LIN {X 0,Y 249.004,Z 314.463,A -85,B 0,C 180,E1 -18940.479,E2 -18940.479} C_VEL
LIN {X 0,Y 248.994,Z 314.49,A -85,B 0,C 180,E1 -18943.762,E2 -18943.762} C_VEL
LIN {X 0,Y 249.907,Z 317.142,A -85,B 0,C 180,E1 -18944.046,E2 -18944.046} C_VEL
LIN {X 0,Y 252.008,Z 319.997,A -85,B 0,C 180,E1 -18944.567,E2 -18944.567} C_VEL
LIN {X 0,Y 261.034,Z 334.136,A -85,B 0,C 180,E1 -18946.731,E2 -18946.731} C_VEL
LIN {X 0,Y 268.672,Z 348.631,A -85,B 0,C 180,E1 -18948.486,E2 -18948.486} C_VEL
LIN {X 0,Y 273.447,Z 359.161,A -85,B 0,C 180,E1 -18949.559,E2 -18949.559} C_VEL
LIN {X 0,Y 270.893,Z 419.37,A -85,B 0,C 180,E1 -18951.127,E2 -18951.127} C_VEL
LIN {X 0,Y 269.96,Z 432.258,A -85,B 0,C 180,E1 -18951.75,E2 -18951.75} C_VEL
LIN {X 0,Y 268.424,Z 444.743,A -85,B 0,C 180,E1 -18952.621,E2 -18952.621} C_VEL
LIN {X 0,Y 266.516,Z 455.493,A -85,B 0,C 180,E1 -18953.608,E2 -18953.608} C_VEL
LIN {X 0,Y 264.431,Z 466.288,A -85,B 0,C 180,E1 -18954.919,E2 -18954.919} C_VEL
LIN {X 0,Y 261.963,Z 477.569,A -85,B 0,C 180,E1 -18956.701,E2 -18956.701} C_VEL
LIN {X 0,Y 259.375,Z 487.065,A -85,B 0,C 180,E1 -18958.562,E2 -18958.562} C_VEL
LIN {X 0,Y 257.027,Z 495.055,A -85,B 0,C 180,E1 -18960.517,E2 -18960.517} C_VEL
LIN {X 0,Y 254.585,Z 502.795,A -85,B 0,C 180,E1 -18962.904,E2 -18962.904} C_VEL
LIN {X 0,Y 252.411,Z 508.966,A -85,B 0,C 180,E1 -18965.315,E2 -18965.315} C_VEL
LIN {X 0,Y 250.814,Z 513.574,A -85,B 0,C 180,E1 -18967.623,E2 -18967.623} C_VEL
LIN {X 0,Y 249.331,Z 517.523,A -85,B 0,C 180,E1 -18970.231,E2 -18970.231} C_VEL
LIN {X 0,Y 248.648,Z 519.417,A -85,B 0,C 180,E1 -18971.887,E2 -18971.887} C_VEL
LIN {X 0,Y 247.809,Z 521.57,A -85,B 0,C 180,E1 -18974.638,E2 -18974.638} C_VEL
LIN {X 0,Y 247.328,Z 522.447,A -85,B 0,C 180,E1 -18976.861,E2 -18976.861} C_VEL
LIN {X 0,Y 247.024,Z 522.665,A -85,B 0,C 180,E1 -18978.514,E2 -18978.514} C_VEL
LIN {X 0,Y 246.927,Z 522.444,A -85,B 0,C 180,E1 -18980.168,E2 -18980.168} C_VEL
LIN {X 0,Y 246.96,Z 521.821,A -85,B 0,C 180,E1 -18981.821,E2 -18981.821} C_VEL
LIN {X 0,Y 247.195,Z 520.115,A -85,B 0,C 180,E1 -18984.326,E2 -18984.326} C_VEL
LIN {X 0,Y 247.479,Z 516.49,A -85,B 0,C 180,E1 -18987.56,E2 -18987.56} C_VEL
LIN {X 0,Y 248.087,Z 512.532,A -85,B 0,C 180,E1 -18990.001,E2 -18990.001} C_VEL
LIN {X 0,Y 248.838,Z 507.454,A -85,B 0,C 180,E1 -18992.429,E2 -18992.429} C_VEL
LIN {X 0,Y 249.967,Z 501.052,A -85,B 0,C 180,E1 -18994.84,E2 -18994.84} C_VEL
LIN {X 0,Y 251.429,Z 493.077,A -85,B 0,C 180,E1 -18997.227,E2 -18997.227} C_VEL
LIN {X 0,Y 252.886,Z 484.949,A -85,B 0,C 180,E1 -18999.196,E2 -18999.196} C_VEL
LIN {X 0,Y 254.516,Z 475.048,A -85,B 0,C 180,E1 -19001.146,E2 -19001.146} C_VEL
LIN {X 0,Y 256.243,Z 463.84,A -85,B 0,C 180,E1 -19002.877,E2 -19002.877} C_VEL
LIN {X 0,Y 257.699,Z 452.872,A -85,B 0,C 180,E1 -19004.209,E2 -19004.209} C_VEL
LIN {X 0,Y 258.85,Z 440.774,A -85,B 0,C 180,E1 -19005.351,E2 -19005.351} C_VEL
LIN {X 0,Y 259.86,Z 428.037,A -85,B 0,C 180,E1 -19006.196,E2 -19006.196} C_VEL
LIN {X 0,Y 260.444,Z 414.653,A -85,B 0,C 180,E1 -19006.763,E2 -19006.763} C_VEL
LIN {X 0,Y 262.544,Z 346.789,A -85,B 0,C 180,E1 -19008.57,E2 -19008.57} C_VEL
LIN {X 0,Y 256.779,Z 331.182,A -85,B 0,C 180,E1 -19009.625,E2 -19009.625} C_VEL
LIN {X 0,Y 249.824,Z 316.729,A -85,B 0,C 180,E1 -19010.835,E2 -19010.835} C_VEL
LIN {X 0,Y 249.109,Z 314.453,A -85,B 0,C 180,E1 -19011.042,E2 -19011.042} C_VEL
LIN {X 0,Y 249.09,Z 314.446,A -85,B 0,C 180,E1 -19015.46,E2 -19015.46} C_VEL
LIN {X 0,Y 249.042,Z 314.462,A -85,B 0,C 180,E1 -19018.974,E2 -19018.974} C_VEL
LIN {X 0,Y 249.032,Z 314.463,A -85,B 0,C 180,E1 -19022.427,E2 -19022.427} C_VEL
LIN {X 0,Y 249.032,Z 314.463,A -85,B 0,C 180,E1 -19026.346,E2 -19026.346} C_VEL
LIN {X 0,Y 248.984,Z 314.465,A -85,B 0,C 180,E1 -19030.484,E2 -19030.484} C_VEL
LIN {X 0,Y 248.967,Z 314.471,A -85,B 0,C 180,E1 -19034.889,E2 -19034.889} C_VEL
LIN {X 0,Y 248.982,Z 314.46,A -85,B 0,C 180,E1 -19037.355,E2 -19037.355} C_VEL
LIN {X 0,Y 249.044,Z 314.459,A -85,B 0,C 180,E1 -19042.202,E2 -19042.202} C_VEL
LIN {X 0,Y 249.048,Z 314.45,A -85,B 0,C 180,E1 -19045.639,E2 -19045.639} C_VEL
LIN {X 0,Y 249.007,Z 314.468,A -85,B 0,C 180,E1 -19049.466,E2 -19049.466} C_VEL
LIN {X 0,Y 249.032,Z 314.458,A -85,B 0,C 180,E1 -19053.157,E2 -19053.157} C_VEL
LIN {X 0,Y 249.049,Z 314.455,A -85,B 0,C 180,E1 -19056.729,E2 -19056.729} C_VEL
LIN {X 0,Y 249.09,Z 314.456,A -85,B 0,C 180,E1 -19060.209,E2 -19060.209} C_VEL
LIN {X 0,Y 249.201,Z 314.431,A -85,B 0,C 180,E1 -19063.619,E2 -19063.619} C_VEL
LIN {X 0,Y 249.238,Z 314.436,A -85,B 0,C 180,E1 -19068.615,E2 -19068.615} C_VEL
LIN {X 0,Y 249.44,Z 314.412,A -85,B 0,C 180,E1 -19071.901,E2 -19071.901} C_VEL
LIN {X 0,Y 249.265,Z 314.416,A -85,B 0,C 180,E1 -19075.147,E2 -19075.147} C_VEL
LIN {X 0,Y 249.661,Z 314.382,A -85,B 0,C 180,E1 -19078.386,E2 -19078.386} C_VEL
LIN {X 0,Y 249.663,Z 314.384,A -85,B 0,C 180,E1 -19081.613,E2 -19081.613} C_VEL
LIN {X 0,Y 249.429,Z 314.398,A -85,B 0,C 180,E1 -19086.471,E2 -19086.471} C_VEL
LIN {X 0,Y 249.37,Z 314.418,A -85,B 0,C 180,E1 -19089.587,E2 -19089.587} C_VEL
LIN {X 0,Y 248.563,Z 314.523,A -85,B 0,C 180,E1 -19090.932,E2 -19090.932} C_VEL
LIN {X 0,Y 245.674,Z 314.891,A -85,B 0,C 180,E1 -19093.126,E2 -19093.126} C_VEL
LIN {X 0,Y 243.279,Z 315.191,A -85,B 0,C 180,E1 -19094.912,E2 -19094.912} C_VEL
LIN {X 0,Y 242.221,Z 315.317,A -85,B 0,C 180,E1 -19096.296,E2 -19096.296} C_VEL
LIN {X 0,Y 242.114,Z 315.327,A -85,B 0,C 180,E1 -19096.766,E2 -19096.766} C_VEL
LIN {X 0,Y 241.996,Z 315.339,A -85,B 0,C 180,E1 -19101.665,E2 -19101.665} C_VEL
LIN {X 0,Y 242.036,Z 315.335,A -85,B 0,C 180,E1 -19105.82,E2 -19105.82} C_VEL
LIN {X 0,Y 241.967,Z 315.344,A -85,B 0,C 180,E1 -19109.588,E2 -19109.588} C_VEL
LIN {X 0,Y 241.982,Z 315.344,A -85,B 0,C 180,E1 -19113.492,E2 -19113.492} C_VEL
LIN {X 0,Y 241.986,Z 315.343,A -85,B 0,C 180,E1 -19117.582,E2 -19117.582} C_VEL
LIN {X 0,Y 241.911,Z 315.351,A -85,B 0,C 180,E1 -19121.928,E2 -19121.928} C_VEL
LIN {X 0,Y 241.903,Z 315.35,A -85,B 0,C 180,E1 -19126.579,E2 -19126.579} C_VEL
LIN {X 0,Y 241.995,Z 315.342,A -85,B 0,C 180,E1 -19131.64,E2 -19131.64} C_VEL
LIN {X 0,Y 242.078,Z 315.472,A -85,B 0,C 180,E1 -19133.376,E2 -19133.376} C_VEL
LIN {X 0,Y 244.407,Z 325.946,A -85,B 0,C 180,E1 -19137.372,E2 -19137.372} C_VEL
LIN {X 0,Y 245.662,Z 332.102,A -85,B 0,C 180,E1 -19139.542,E2 -19139.542} C_VEL
LIN {X 0,Y 250.101,Z 344.165,A -85,B 0,C 180,E1 -19140.425,E2 -19140.425} C_VEL
LIN {X 0,Y 253.396,Z 369.809,A -85,B 0,C 180,E1 -19141.569,E2 -19141.569} C_VEL
LIN {X 0,Y 255.075,Z 385.817,A -85,B 0,C 180,E1 -19142.225,E2 -19142.225} C_VEL
LIN {X 0,Y 253.455,Z 440.891,A -85,B 0,C 180,E1 -19143.772,E2 -19143.772} C_VEL
LIN {X 0,Y 252.408,Z 454.202,A -85,B 0,C 180,E1 -19144.431,E2 -19144.431} C_VEL
LIN {X 0,Y 250.993,Z 466.976,A -85,B 0,C 180,E1 -19145.384,E2 -19145.384} C_VEL
LIN {X 0,Y 249.503,Z 478.329,A -85,B 0,C 180,E1 -19146.554,E2 -19146.554} C_VEL
LIN {X 0,Y 247.677,Z 490.055,A -85,B 0,C 180,E1 -19148.133,E2 -19148.133} C_VEL
LIN {X 0,Y 245.777,Z 500.589,A -85,B 0,C 180,E1 -19149.931,E2 -19149.931} C_VEL
LIN {X 0,Y 244.087,Z 510.234,A -85,B 0,C 180,E1 -19152.01,E2 -19152.01} C_VEL
LIN {X 0,Y 243.125,Z 516.416,A -85,B 0,C 180,E1 -19153.629,E2 -19153.629} C_VEL
LIN {X 0,Y 241.768,Z 524.334,A -85,B 0,C 180,E1 -19156.123,E2 -19156.123} C_VEL
LIN {X 0,Y 240.881,Z 529.707,A -85,B 0,C 180,E1 -19158.214,E2 -19158.214} C_VEL
LIN {X 0,Y 240.312,Z 534.946,A -85,B 0,C 180,E1 -19160.743,E2 -19160.743} C_VEL
LIN {X 0,Y 239.98,Z 538.995,A -85,B 0,C 180,E1 -19163.272,E2 -19163.272} C_VEL
LIN {X 0,Y 239.92,Z 541.078,A -85,B 0,C 180,E1 -19164.957,E2 -19164.957} C_VEL
LIN {X 0,Y 239.949,Z 542.73,A -85,B 0,C 180,E1 -19166.641,E2 -19166.641} C_VEL
LIN {X 0,Y 239.999,Z 543.969,A -85,B 0,C 180,E1 -19168.321,E2 -19168.321} C_VEL
LIN {X 0,Y 240.02,Z 544.783,A -85,B 0,C 180,E1 -19169.999,E2 -19169.999} C_VEL
LIN {X 0,Y 239.975,Z 545.159,A -85,B 0,C 180,E1 -19171.677,E2 -19171.677} C_VEL
LIN {X 0,Y 239.843,Z 544.771,A -85,B 0,C 180,E1 -19174.94,E2 -19174.94} C_VEL
LIN {X 0,Y 239.9,Z 543.946,A -85,B 0,C 180,E1 -19176.728,E2 -19176.728} C_VEL
LIN {X 0,Y 240.161,Z 542.72,A -85,B 0,C 180,E1 -19178.413,E2 -19178.413} C_VEL
LIN {X 0,Y 241.118,Z 539.053,A -85,B 0,C 180,E1 -19181.772,E2 -19181.772} C_VEL
LIN {X 0,Y 242.269,Z 535.123,A -85,B 0,C 180,E1 -19184.274,E2 -19184.274} C_VEL
LIN {X 0,Y 244.025,Z 530.087,A -85,B 0,C 180,E1 -19186.737,E2 -19186.737} C_VEL
LIN {X 0,Y 246.049,Z 523.992,A -85,B 0,C 180,E1 -19189.098,E2 -19189.098} C_VEL
LIN {X 0,Y 248.08,Z 517.373,A -85,B 0,C 180,E1 -19191.173,E2 -19191.173} C_VEL
LIN {X 0,Y 250.476,Z 509.699,A -85,B 0,C 180,E1 -19193.129,E2 -19193.129} C_VEL
LIN {X 0,Y 253.26,Z 500.391,A -85,B 0,C 180,E1 -19195.035,E2 -19195.035} C_VEL
LIN {X 0,Y 256.042,Z 490.065,A -85,B 0,C 180,E1 -19196.709,E2 -19196.709} C_VEL
LIN {X 0,Y 258.723,Z 478.628,A -85,B 0,C 180,E1 -19198.162,E2 -19198.162} C_VEL
LIN {X 0,Y 261.046,Z 466.681,A -85,B 0,C 180,E1 -19199.317,E2 -19199.317} C_VEL
LIN {X 0,Y 263.056,Z 453.416,A -85,B 0,C 180,E1 -19200.227,E2 -19200.227} C_VEL
LIN {X 0,Y 264.375,Z 440.684,A -85,B 0,C 180,E1 -19200.81,E2 -19200.81} C_VEL
LIN {X 0,Y 266.485,Z 389.159,A -85,B 0,C 180,E1 -19202.213,E2 -19202.213} C_VEL
LIN {X 0,Y 263.336,Z 367.774,A -85,B 0,C 180,E1 -19203.42,E2 -19203.42} C_VEL
LIN {X 0,Y 262.236,Z 363.038,A -85,B 0,C 180,E1 -19203.76,E2 -19203.76} C_VEL
LIN {X 0,Y 255.3,Z 347.85,A -85,B 0,C 180,E1 -19205.488,E2 -19205.488} C_VEL
LIN {X 0,Y 248.566,Z 334.814,A -85,B 0,C 180,E1 -19207.241,E2 -19207.241} C_VEL
LIN {X 0,Y 246.197,Z 330.21,A -85,B 0,C 180,E1 -19207.947,E2 -19207.947} C_VEL
LIN {X 0,Y 243.761,Z 321.533,A -85,B 0,C 180,E1 -19211.966,E2 -19211.966} C_VEL
LIN {X 0,Y 241.952,Z 315.348,A -85,B 0,C 180,E1 -19215.109,E2 -19215.109} C_VEL
LIN {X 0,Y 241.928,Z 315.343,A -85,B 0,C 180,E1 -19219.05,E2 -19219.05} C_VEL
LIN {X 0,Y 241.986,Z 315.335,A -85,B 0,C 180,E1 -19222.418,E2 -19222.418} C_VEL
LIN {X 0,Y 241.977,Z 315.34,A -85,B 0,C 180,E1 -19226.507,E2 -19226.507} C_VEL
LIN {X 0,Y 242.032,Z 315.334,A -85,B 0,C 180,E1 -19230.587,E2 -19230.587} C_VEL
LIN {X 0,Y 242.064,Z 315.331,A -85,B 0,C 180,E1 -19234.183,E2 -19234.183} C_VEL
LIN {X 0,Y 242.05,Z 315.332,A -85,B 0,C 180,E1 -19238.297,E2 -19238.297} C_VEL
LIN {X 0,Y 242.159,Z 315.311,A -85,B 0,C 180,E1 -19243.278,E2 -19243.278} C_VEL
LIN {X 0,Y 242.183,Z 315.308,A -85,B 0,C 180,E1 -19248.28,E2 -19248.28} C_VEL
LIN {X 0,Y 242.432,Z 315.277,A -85,B 0,C 180,E1 -19251.666,E2 -19251.666} C_VEL
LIN {X 0,Y 242.258,Z 315.304,A -85,B 0,C 180,E1 -19255.008,E2 -19255.008} C_VEL
LIN {X 0,Y 242.634,Z 315.26,A -85,B 0,C 180,E1 -19258.341,E2 -19258.341} C_VEL
LIN {X 0,Y 242.634,Z 315.256,A -85,B 0,C 180,E1 -19261.66,E2 -19261.66} C_VEL
LIN {X 0,Y 242.427,Z 315.284,A -85,B 0,C 180,E1 -19266.733,E2 -19266.733} C_VEL
LIN {X 0,Y 242.343,Z 315.291,A -85,B 0,C 180,E1 -19270.021,E2 -19270.021} C_VEL
LIN {X 0,Y 242.164,Z 315.319,A -85,B 0,C 180,E1 -19275.142,E2 -19275.142} C_VEL
LIN {X 0,Y 242.071,Z 315.327,A -85,B 0,C 180,E1 -19278.625,E2 -19278.625} C_VEL
LIN {X 0,Y 242.011,Z 315.333,A -85,B 0,C 180,E1 -19282.181,E2 -19282.181} C_VEL
LIN {X 0,Y 242.064,Z 315.326,A -85,B 0,C 180,E1 -19285.839,E2 -19285.839} C_VEL
LIN {X 0,Y 242.005,Z 315.334,A -85,B 0,C 180,E1 -19289.584,E2 -19289.584} C_VEL
LIN {X 0,Y 241.979,Z 315.34,A -85,B 0,C 180,E1 -19293.494,E2 -19293.494} C_VEL
LIN {X 0,Y 241.987,Z 315.336,A -85,B 0,C 180,E1 -19297.583,E2 -19297.583} C_VEL
LIN {X 0,Y 241.953,Z 315.364,A -85,B 0,C 180,E1 -19302.306,E2 -19302.306} C_VEL
LIN {X 0,Y 242.979,Z 318.216,A -85,B 0,C 180,E1 -19302.644,E2 -19302.644} C_VEL
LIN {X 0,Y 244.901,Z 320.584,A -85,B 0,C 180,E1 -19303.147,E2 -19303.147} C_VEL
LIN {X 0,Y 247.13,Z 324.018,A -85,B 0,C 180,E1 -19303.743,E2 -19303.743} C_VEL
LIN {X 0,Y 255.301,Z 336.912,A -85,B 0,C 180,E1 -19305.805,E2 -19305.805} C_VEL
LIN {X 0,Y 260.026,Z 345.326,A -85,B 0,C 180,E1 -19306.943,E2 -19306.943} C_VEL
LIN {X 0,Y 266.261,Z 358.237,A -85,B 0,C 180,E1 -19308.418,E2 -19308.418} C_VEL
LIN {X 0,Y 267.602,Z 361.247,A -85,B 0,C 180,E1 -19308.73,E2 -19308.73} C_VEL
LIN {X 0,Y 265.096,Z 418.751,A -85,B 0,C 180,E1 -19310.249,E2 -19310.249} C_VEL
LIN {X 0,Y 264.104,Z 431.812,A -85,B 0,C 180,E1 -19310.865,E2 -19310.865} C_VEL
LIN {X 0,Y 262.551,Z 444.507,A -85,B 0,C 180,E1 -19311.757,E2 -19311.757} C_VEL
LIN {X 0,Y 260.382,Z 456.275,A -85,B 0,C 180,E1 -19312.85,E2 -19312.85} C_VEL
LIN {X 0,Y 257.948,Z 468.272,A -85,B 0,C 180,E1 -19314.383,E2 -19314.383} C_VEL
LIN {X 0,Y 255.306,Z 479.371,A -85,B 0,C 180,E1 -19316.214,E2 -19316.214} C_VEL
LIN {X 0,Y 252.698,Z 488.496,A -85,B 0,C 180,E1 -19318.102,E2 -19318.102} C_VEL
LIN {X 0,Y 249.907,Z 497.336,A -85,B 0,C 180,E1 -19320.418,E2 -19320.418} C_VEL
LIN {X 0,Y 247.325,Z 504.959,A -85,B 0,C 180,E1 -19322.958,E2 -19322.958} C_VEL
LIN {X 0,Y 245.182,Z 510.763,A -85,B 0,C 180,E1 -19325.442,E2 -19325.442} C_VEL
LIN {X 0,Y 243.46,Z 515.287,A -85,B 0,C 180,E1 -19327.96,E2 -19327.96} C_VEL
LIN {X 0,Y 242.52,Z 517.656,A -85,B 0,C 180,E1 -19329.651,E2 -19329.651} C_VEL
LIN {X 0,Y 241.743,Z 519.584,A -85,B 0,C 180,E1 -19331.351,E2 -19331.351} C_VEL
LIN {X 0,Y 240.774,Z 521.944,A -85,B 0,C 180,E1 -19334.42,E2 -19334.42} C_VEL
LIN {X 0,Y 240.299,Z 522.737,A -85,B 0,C 180,E1 -19336.47,E2 -19336.47} C_VEL
LIN {X 0,Y 239.979,Z 522.985,A -85,B 0,C 180,E1 -19338.172,E2 -19338.172} C_VEL
LIN {X 0,Y 239.851,Z 522.823,A -85,B 0,C 180,E1 -19339.875,E2 -19339.875} C_VEL
LIN {X 0,Y 239.969,Z 521.251,A -85,B 0,C 180,E1 -19343.274,E2 -19343.274} C_VEL
LIN {X 0,Y 240.124,Z 519.885,A -85,B 0,C 180,E1 -19344.964,E2 -19344.964} C_VEL
LIN {X 0,Y 240.385,Z 517.019,A -85,B 0,C 180,E1 -19347.488,E2 -19347.488} C_VEL
LIN {X 0,Y 241.009,Z 513.127,A -85,B 0,C 180,E1 -19350.001,E2 -19350.001} C_VEL
LIN {X 0,Y 241.771,Z 508.125,A -85,B 0,C 180,E1 -19352.5,E2 -19352.5} C_VEL
LIN {X 0,Y 242.92,Z 501.834,A -85,B 0,C 180,E1 -19354.98,E2 -19354.98} C_VEL
LIN {X 0,Y 244.426,Z 493.956,A -85,B 0,C 180,E1 -19357.435,E2 -19357.435} C_VEL
LIN {X 0,Y 246.221,Z 484.171,A -85,B 0,C 180,E1 -19359.862,E2 -19359.862} C_VEL
LIN {X 0,Y 247.986,Z 473.94,A -85,B 0,C 180,E1 -19361.858,E2 -19361.858} C_VEL
LIN {X 0,Y 249.805,Z 462.389,A -85,B 0,C 180,E1 -19363.629,E2 -19363.629} C_VEL
LIN {X 0,Y 251.284,Z 450.994,A -85,B 0,C 180,E1 -19364.994,E2 -19364.994} C_VEL
LIN {X 0,Y 252.442,Z 439.229,A -85,B 0,C 180,E1 -19366.062,E2 -19366.062} C_VEL
LIN {X 0,Y 253.443,Z 425.644,A -85,B 0,C 180,E1 -19366.929,E2 -19366.929} C_VEL
LIN {X 0,Y 253.951,Z 413.482,A -85,B 0,C 180,E1 -19367.413,E2 -19367.413} C_VEL
LIN {X 0,Y 256.048,Z 348.219,A -85,B 0,C 180,E1 -19369.183,E2 -19369.183} C_VEL
LIN {X 0,Y 250.573,Z 333.661,A -85,B 0,C 180,E1 -19370.219,E2 -19370.219} C_VEL
LIN {X 0,Y 243.192,Z 318.383,A -85,B 0,C 180,E1 -19371.559,E2 -19371.559} C_VEL
LIN {X 0,Y 242.026,Z 315.332,A -85,B 0,C 180,E1 -19371.839,E2 -19371.839} C_VEL
LIN {X 0,Y 242.037,Z 315.326,A -85,B 0,C 180,E1 -19375.822,E2 -19375.822} C_VEL
LIN {X 0,Y 241.974,Z 315.342,A -85,B 0,C 180,E1 -19379.589,E2 -19379.589} C_VEL
LIN {X 0,Y 241.984,Z 315.342,A -85,B 0,C 180,E1 -19383.493,E2 -19383.493} C_VEL
LIN {X 0,Y 241.988,Z 315.342,A -85,B 0,C 180,E1 -19387.583,E2 -19387.583} C_VEL
LIN {X 0,Y 241.913,Z 315.345,A -85,B 0,C 180,E1 -19391.929,E2 -19391.929} C_VEL
LIN {X 0,Y 241.904,Z 315.345,A -85,B 0,C 180,E1 -19396.58,E2 -19396.58} C_VEL
LIN {X 0,Y 241.989,Z 315.341,A -85,B 0,C 180,E1 -19401.644,E2 -19401.644} C_VEL
LIN {X 0,Y 241.979,Z 315.332,A -85,B 0,C 180,E1 -19404.487,E2 -19404.487} C_VEL
LIN {X 0,Y 241.958,Z 315.343,A -85,B 0,C 180,E1 -19408.477,E2 -19408.477} C_VEL
LIN {X 0,Y 241.969,Z 315.337,A -85,B 0,C 180,E1 -19412.307,E2 -19412.307} C_VEL
LIN {X 0,Y 242.014,Z 315.327,A -85,B 0,C 180,E1 -19416.011,E2 -19416.011} C_VEL
LIN {X 0,Y 242.026,Z 315.337,A -85,B 0,C 180,E1 -19419.606,E2 -19419.606} C_VEL
LIN {X 0,Y 242.133,Z 315.314,A -85,B 0,C 180,E1 -19423.307,E2 -19423.307} C_VEL
LIN {X 0,Y 242.172,Z 315.318,A -85,B 0,C 180,E1 -19428.279,E2 -19428.279} C_VEL
LIN {X 0,Y 242.39,Z 315.29,A -85,B 0,C 180,E1 -19431.664,E2 -19431.664} C_VEL
LIN {X 0,Y 242.406,Z 315.281,A -85,B 0,C 180,E1 -19433.34,E2 -19433.34} C_VEL
LIN {X 0,Y 242.621,Z 315.257,A -85,B 0,C 180,E1 -19438.34,E2 -19438.34} C_VEL
LIN {X 0,Y 242.623,Z 315.261,A -85,B 0,C 180,E1 -19441.659,E2 -19441.659} C_VEL
LIN {X 0,Y 242.4,Z 315.273,A -85,B 0,C 180,E1 -19446.659,E2 -19446.659} C_VEL
LIN {X 0,Y 242.27,Z 315.303,A -85,B 0,C 180,E1 -19450.023,E2 -19450.023} C_VEL
LIN {X 0,Y 242.131,Z 315.323,A -85,B 0,C 180,E1 -19455.143,E2 -19455.143} C_VEL
LIN {X 0,Y 242.114,Z 315.327,A -85,B 0,C 180,E1 -19456.766,E2 -19456.766} C_VEL
LIN {X 0,Y 241.369,Z 315.417,A -85,B 0,C 180,E1 -19458.154,E2 -19458.154} C_VEL
LIN {X 0,Y 238.435,Z 315.785,A -85,B 0,C 180,E1 -19460.416,E2 -19460.416} C_VEL
LIN {X 0,Y 236.002,Z 316.087,A -85,B 0,C 180,E1 -19462.259,E2 -19462.259} C_VEL
LIN {X 0,Y 234.992,Z 316.212,A -85,B 0,C 180,E1 -19463.691,E2 -19463.691} C_VEL
LIN {X 0,Y 234.925,Z 316.22,A -85,B 0,C 180,E1 -19464.176,E2 -19464.176} C_VEL
LIN {X 0,Y 234.946,Z 316.219,A -85,B 0,C 180,E1 -19466.66,E2 -19466.66} C_VEL
LIN {X 0,Y 234.898,Z 316.226,A -85,B 0,C 180,E1 -19470.572,E2 -19470.572} C_VEL
LIN {X 0,Y 234.928,Z 316.223,A -85,B 0,C 180,E1 -19474.638,E2 -19474.638} C_VEL
LIN {X 0,Y 234.914,Z 316.225,A -85,B 0,C 180,E1 -19478.934,E2 -19478.934} C_VEL
LIN {X 0,Y 234.856,Z 316.232,A -85,B 0,C 180,E1 -19483.493,E2 -19483.493} C_VEL
LIN {X 0,Y 234.856,Z 316.227,A -85,B 0,C 180,E1 -19486.505,E2 -19486.505} C_VEL
LIN {X 0,Y 234.92,Z 316.224,A -85,B 0,C 180,E1 -19491.078,E2 -19491.078} C_VEL
LIN {X 0,Y 234.996,Z 316.343,A -85,B 0,C 180,E1 -19492.726,E2 -19492.726} C_VEL
LIN {X 0,Y 236.957,Z 324.925,A -85,B 0,C 180,E1 -19496.146,E2 -19496.146} C_VEL
LIN {X 0,Y 238.377,Z 331.628,A -85,B 0,C 180,E1 -19498.654,E2 -19498.654} C_VEL
LIN {X 0,Y 243.925,Z 346.675,A -85,B 0,C 180,E1 -19499.81,E2 -19499.81} C_VEL
LIN {X 0,Y 246.998,Z 371.172,A -85,B 0,C 180,E1 -19500.936,E2 -19500.936} C_VEL
LIN {X 0,Y 248.563,Z 386.873,A -85,B 0,C 180,E1 -19501.595,E2 -19501.595} C_VEL
LIN {X 0,Y 246.918,Z 440.487,A -85,B 0,C 180,E1 -19503.137,E2 -19503.137} C_VEL
LIN {X 0,Y 245.853,Z 453.828,A -85,B 0,C 180,E1 -19503.812,E2 -19503.812} C_VEL
LIN {X 0,Y 244.402,Z 466.616,A -85,B 0,C 180,E1 -19504.788,E2 -19504.788} C_VEL
LIN {X 0,Y 242.713,Z 478.774,A -85,B 0,C 180,E1 -19506.084,E2 -19506.084} C_VEL
LIN {X 0,Y 240.829,Z 490.358,A -85,B 0,C 180,E1 -19507.704,E2 -19507.704} C_VEL
LIN {X 0,Y 238.881,Z 500.782,A -85,B 0,C 180,E1 -19509.55,E2 -19509.55} C_VEL
LIN {X 0,Y 237.309,Z 509.477,A -85,B 0,C 180,E1 -19511.478,E2 -19511.478} C_VEL
LIN {X 0,Y 236.304,Z 515.701,A -85,B 0,C 180,E1 -19513.142,E2 -19513.142} C_VEL
LIN {X 0,Y 234.858,Z 523.708,A -85,B 0,C 180,E1 -19515.706,E2 -19515.706} C_VEL
LIN {X 0,Y 233.878,Z 529.113,A -85,B 0,C 180,E1 -19517.856,E2 -19517.856} C_VEL
LIN {X 0,Y 233.26,Z 534.412,A -85,B 0,C 180,E1 -19520.46,E2 -19520.46} C_VEL
LIN {X 0,Y 232.904,Z 538.51,A -85,B 0,C 180,E1 -19523.066,E2 -19523.066} C_VEL
LIN {X 0,Y 232.841,Z 540.747,A -85,B 0,C 180,E1 -19524.914,E2 -19524.914} C_VEL
LIN {X 0,Y 232.927,Z 543.568,A -85,B 0,C 180,E1 -19528.27,E2 -19528.27} C_VEL
LIN {X 0,Y 232.948,Z 544.417,A -85,B 0,C 180,E1 -19529.999,E2 -19529.999} C_VEL
LIN {X 0,Y 232.902,Z 544.819,A -85,B 0,C 180,E1 -19531.728,E2 -19531.728} C_VEL
LIN {X 0,Y 232.764,Z 544.439,A -85,B 0,C 180,E1 -19535.196,E2 -19535.196} C_VEL
LIN {X 0,Y 232.821,Z 543.673,A -85,B 0,C 180,E1 -19536.934,E2 -19536.934} C_VEL
LIN {X 0,Y 233.109,Z 542.481,A -85,B 0,C 180,E1 -19538.669,E2 -19538.669} C_VEL
LIN {X 0,Y 234.134,Z 538.858,A -85,B 0,C 180,E1 -19542.128,E2 -19542.128} C_VEL
LIN {X 0,Y 235.375,Z 534.973,A -85,B 0,C 180,E1 -19544.701,E2 -19544.701} C_VEL
LIN {X 0,Y 237.19,Z 529.987,A -85,B 0,C 180,E1 -19547.235,E2 -19547.235} C_VEL
LIN {X 0,Y 239.675,Z 522.86,A -85,B 0,C 180,E1 -19550.044,E2 -19550.044} C_VEL
LIN {X 0,Y 242.401,Z 514.502,A -85,B 0,C 180,E1 -19552.591,E2 -19552.591} C_VEL
LIN {X 0,Y 245.099,Z 506.308,A -85,B 0,C 180,E1 -19554.567,E2 -19554.567} C_VEL
LIN {X 0,Y 248.093,Z 496.337,A -85,B 0,C 180,E1 -19556.497,E2 -19556.497} C_VEL
LIN {X 0,Y 251.097,Z 485.084,A -85,B 0,C 180,E1 -19558.184,E2 -19558.184} C_VEL
LIN {X 0,Y 253.596,Z 474.083,A -85,B 0,C 180,E1 -19559.465,E2 -19559.465} C_VEL
LIN {X 0,Y 255.897,Z 461.901,A -85,B 0,C 180,E1 -19560.535,E2 -19560.535} C_VEL
LIN {X 0,Y 257.7,Z 448.878,A -85,B 0,C 180,E1 -19561.339,E2 -19561.339} C_VEL
LIN {X 0,Y 258.819,Z 435.274,A -85,B 0,C 180,E1 -19561.874,E2 -19561.874} C_VEL
LIN {X 0,Y 260.742,Z 390.727,A -85,B 0,C 180,E1 -19563.07,E2 -19563.07} C_VEL
LIN {X 0,Y 258.298,Z 373.078,A -85,B 0,C 180,E1 -19564.079,E2 -19564.079} C_VEL
LIN {X 0,Y 257.011,Z 366.357,A -85,B 0,C 180,E1 -19564.533,E2 -19564.533} C_VEL
LIN {X 0,Y 249.894,Z 350.731,A -85,B 0,C 180,E1 -19566.391,E2 -19566.391} C_VEL
LIN {X 0,Y 243.803,Z 338.95,A -85,B 0,C 180,E1 -19568.053,E2 -19568.053} C_VEL
LIN {X 0,Y 241.067,Z 334.042,A -85,B 0,C 180,E1 -19568.827,E2 -19568.827} C_VEL
LIN {X 0,Y 238.84,Z 329.792,A -85,B 0,C 180,E1 -19569.526,E2 -19569.526} C_VEL
LIN {X 0,Y 236.48,Z 321.57,A -85,B 0,C 180,E1 -19573.574,E2 -19573.574} C_VEL
LIN {X 0,Y 234.877,Z 316.222,A -85,B 0,C 180,E1 -19576.512,E2 -19576.512} C_VEL
LIN {X 0,Y 234.915,Z 316.22,A -85,B 0,C 180,E1 -19581.078,E2 -19581.078} C_VEL
LIN {X 0,Y 234.927,Z 316.212,A -85,B 0,C 180,E1 -19585.362,E2 -19585.362} C_VEL
LIN {X 0,Y 234.927,Z 316.215,A -85,B 0,C 180,E1 -19589.432,E2 -19589.432} C_VEL
LIN {X 0,Y 234.99,Z 316.211,A -85,B 0,C 180,E1 -19593.794,E2 -19593.794} C_VEL
LIN {X 0,Y 235.008,Z 316.202,A -85,B 0,C 180,E1 -19598.97,E2 -19598.97} C_VEL
LIN {X 0,Y 235.093,Z 316.192,A -85,B 0,C 180,E1 -19603.059,E2 -19603.059} C_VEL
LIN {X 0,Y 235.127,Z 316.197,A -85,B 0,C 180,E1 -19606.166,E2 -19606.166} C_VEL
LIN {X 0,Y 235.387,Z 316.156,A -85,B 0,C 180,E1 -19611.415,E2 -19611.415} C_VEL
LIN {X 0,Y 235.402,Z 316.157,A -85,B 0,C 180,E1 -19613.142,E2 -19613.142} C_VEL
LIN {X 0,Y 235.593,Z 316.137,A -85,B 0,C 180,E1 -19618.291,E2 -19618.291} C_VEL
LIN {X 0,Y 235.593,Z 316.133,A -85,B 0,C 180,E1 -19621.71,E2 -19621.71} C_VEL
LIN {X 0,Y 235.403,Z 316.161,A -85,B 0,C 180,E1 -19626.859,E2 -19626.859} C_VEL
LIN {X 0,Y 235.25,Z 316.176,A -85,B 0,C 180,E1 -19630.326,E2 -19630.326} C_VEL
LIN {X 0,Y 235.111,Z 316.198,A -85,B 0,C 180,E1 -19635.607,E2 -19635.607} C_VEL
LIN {X 0,Y 235.006,Z 316.211,A -85,B 0,C 180,E1 -19639.206,E2 -19639.206} C_VEL
LIN {X 0,Y 234.959,Z 316.216,A -85,B 0,C 180,E1 -19642.884,E2 -19642.884} C_VEL
LIN {X 0,Y 234.966,Z 316.215,A -85,B 0,C 180,E1 -19646.658,E2 -19646.658} C_VEL
LIN {X 0,Y 234.92,Z 316.221,A -85,B 0,C 180,E1 -19650.57,E2 -19650.57} C_VEL
LIN {X 0,Y 234.928,Z 316.216,A -85,B 0,C 180,E1 -19654.639,E2 -19654.639} C_VEL
LIN {X 0,Y 234.94,Z 316.213,A -85,B 0,C 180,E1 -19658.946,E2 -19658.946} C_VEL
LIN {X 0,Y 234.895,Z 316.22,A -85,B 0,C 180,E1 -19660.705,E2 -19660.705} C_VEL
LIN {X 0,Y 235.921,Z 319.13,A -85,B 0,C 180,E1 -19661.084,E2 -19661.084} C_VEL
LIN {X 0,Y 238.055,Z 321.599,A -85,B 0,C 180,E1 -19661.682,E2 -19661.682} C_VEL
LIN {X 0,Y 240.192,Z 324.893,A -85,B 0,C 180,E1 -19662.298,E2 -19662.298} C_VEL
LIN {X 0,Y 248.569,Z 337.793,A -85,B 0,C 180,E1 -19664.552,E2 -19664.552} C_VEL
LIN {X 0,Y 254.628,Z 348.265,A -85,B 0,C 180,E1 -19666.087,E2 -19666.087} C_VEL
LIN {X 0,Y 261.078,Z 361.737,A -85,B 0,C 180,E1 -19667.685,E2 -19667.685} C_VEL
LIN {X 0,Y 261.812,Z 363.458,A -85,B 0,C 180,E1 -19667.866,E2 -19667.866} C_VEL
LIN {X 0,Y 259.259,Z 419.591,A -85,B 0,C 180,E1 -19669.379,E2 -19669.379} C_VEL
LIN {X 0,Y 258.219,Z 432.619,A -85,B 0,C 180,E1 -19670.019,E2 -19670.019} C_VEL
LIN {X 0,Y 256.541,Z 445.449,A -85,B 0,C 180,E1 -19670.945,E2 -19670.945} C_VEL
LIN {X 0,Y 254.296,Z 457.063,A -85,B 0,C 180,E1 -19672.055,E2 -19672.055} C_VEL
LIN {X 0,Y 251.755,Z 468.945,A -85,B 0,C 180,E1 -19673.616,E2 -19673.616} C_VEL
LIN {X 0,Y 249.234,Z 479.16,A -85,B 0,C 180,E1 -19675.334,E2 -19675.334} C_VEL
LIN {X 0,Y 246.548,Z 488.186,A -85,B 0,C 180,E1 -19677.208,E2 -19677.208} C_VEL
LIN {X 0,Y 243.921,Z 496.222,A -85,B 0,C 180,E1 -19679.291,E2 -19679.291} C_VEL
LIN {X 0,Y 241.314,Z 503.742,A -85,B 0,C 180,E1 -19681.755,E2 -19681.755} C_VEL
LIN {X 0,Y 238.59,Z 510.77,A -85,B 0,C 180,E1 -19684.716,E2 -19684.716} C_VEL
LIN {X 0,Y 236.742,Z 515.378,A -85,B 0,C 180,E1 -19687.3,E2 -19687.3} C_VEL
LIN {X 0,Y 235.736,Z 517.789,A -85,B 0,C 180,E1 -19689.039,E2 -19689.039} C_VEL
LIN {X 0,Y 234.882,Z 519.75,A -85,B 0,C 180,E1 -19690.785,E2 -19690.785} C_VEL
LIN {X 0,Y 234.227,Z 521.285,A -85,B 0,C 180,E1 -19692.54,E2 -19692.54} C_VEL
LIN {X 0,Y 233.709,Z 522.362,A -85,B 0,C 180,E1 -19694.299,E2 -19694.299} C_VEL
LIN {X 0,Y 233.28,Z 523.026,A -85,B 0,C 180,E1 -19696.055,E2 -19696.055} C_VEL
LIN {X 0,Y 232.793,Z 523.189,A -85,B 0,C 180,E1 -19699.565,E2 -19699.565} C_VEL
LIN {X 0,Y 232.77,Z 522.638,A -85,B 0,C 180,E1 -19701.318,E2 -19701.318} C_VEL
LIN {X 0,Y 233.032,Z 520.678,A -85,B 0,C 180,E1 -19704.42,E2 -19704.42} C_VEL
LIN {X 0,Y 233.294,Z 517.547,A -85,B 0,C 180,E1 -19707.411,E2 -19707.411} C_VEL
LIN {X 0,Y 233.929,Z 513.721,A -85,B 0,C 180,E1 -19710.001,E2 -19710.001} C_VEL
LIN {X 0,Y 234.705,Z 508.789,A -85,B 0,C 180,E1 -19712.575,E2 -19712.575} C_VEL
LIN {X 0,Y 235.873,Z 502.589,A -85,B 0,C 180,E1 -19715.129,E2 -19715.129} C_VEL
LIN {X 0,Y 237.399,Z 494.84,A -85,B 0,C 180,E1 -19717.657,E2 -19717.657} C_VEL
LIN {X 0,Y 239.257,Z 485.162,A -85,B 0,C 180,E1 -19720.152,E2 -19720.152} C_VEL
LIN {X 0,Y 241.089,Z 475.138,A -85,B 0,C 180,E1 -19722.202,E2 -19722.202} C_VEL
LIN {X 0,Y 242.952,Z 463.777,A -85,B 0,C 180,E1 -19724.021,E2 -19724.021} C_VEL
LIN {X 0,Y 244.514,Z 452.643,A -85,B 0,C 180,E1 -19725.42,E2 -19725.42} C_VEL
LIN {X 0,Y 245.681,Z 441.411,A -85,B 0,C 180,E1 -19726.517,E2 -19726.517} C_VEL
LIN {X 0,Y 246.746,Z 428.675,A -85,B 0,C 180,E1 -19727.403,E2 -19727.403} C_VEL
LIN {X 0,Y 247.397,Z 415.273,A -85,B 0,C 180,E1 -19727.996,E2 -19727.996} C_VEL
LIN {X 0,Y 249.692,Z 350.118,A -85,B 0,C 180,E1 -19729.8,E2 -19729.8} C_VEL
LIN {X 0,Y 244.479,Z 336.371,A -85,B 0,C 180,E1 -19730.823,E2 -19730.823} C_VEL
LIN {X 0,Y 237.593,Z 322.121,A -85,B 0,C 180,E1 -19732.127,E2 -19732.127} C_VEL
LIN {X 0,Y 235.094,Z 317.005,A -85,B 0,C 180,E1 -19732.622,E2 -19732.622} C_VEL
LIN {X 0,Y 234.958,Z 316.214,A -85,B 0,C 180,E1 -19732.682,E2 -19732.682} C_VEL
LIN {X 0,Y 234.95,Z 316.212,A -85,B 0,C 180,E1 -19736.661,E2 -19736.661} C_VEL
LIN {X 0,Y 234.904,Z 316.223,A -85,B 0,C 180,E1 -19740.573,E2 -19740.573} C_VEL
LIN {X 0,Y 234.93,Z 316.221,A -85,B 0,C 180,E1 -19744.639,E2 -19744.639} C_VEL
LIN {X 0,Y 234.917,Z 316.223,A -85,B 0,C 180,E1 -19748.935,E2 -19748.935} C_VEL
LIN {X 0,Y 234.858,Z 316.23,A -85,B 0,C 180,E1 -19753.494,E2 -19753.494} C_VEL
LIN {X 0,Y 234.857,Z 316.222,A -85,B 0,C 180,E1 -19756.506,E2 -19756.506} C_VEL
LIN {X 0,Y 234.923,Z 316.22,A -85,B 0,C 180,E1 -19761.079,E2 -19761.079} C_VEL
LIN {X 0,Y 234.927,Z 316.207,A -85,B 0,C 180,E1 -19765.361,E2 -19765.361} C_VEL
LIN {X 0,Y 234.904,Z 316.224,A -85,B 0,C 180,E1 -19769.428,E2 -19769.428} C_VEL
LIN {X 0,Y 234.95,Z 316.202,A -85,B 0,C 180,E1 -19773.818,E2 -19773.818} C_VEL
LIN {X 0,Y 234.994,Z 316.211,A -85,B 0,C 180,E1 -19778.968,E2 -19778.968} C_VEL
LIN {X 0,Y 235.069,Z 316.194,A -85,B 0,C 180,E1 -19783.086,E2 -19783.086} C_VEL
LIN {X 0,Y 235.105,Z 316.194,A -85,B 0,C 180,E1 -19787.921,E2 -19787.921} C_VEL
LIN {X 0,Y 235.324,Z 316.169,A -85,B 0,C 180,E1 -19791.412,E2 -19791.412} C_VEL
LIN {X 0,Y 235.358,Z 316.158,A -85,B 0,C 180,E1 -19793.14,E2 -19793.14} C_VEL
LIN {X 0,Y 235.581,Z 316.133,A -85,B 0,C 180,E1 -19798.29,E2 -19798.29} C_VEL
LIN {X 0,Y 235.581,Z 316.138,A -85,B 0,C 180,E1 -19801.709,E2 -19801.709} C_VEL
LIN {X 0,Y 235.351,Z 316.151,A -85,B 0,C 180,E1 -19806.86,E2 -19806.86} C_VEL
LIN {X 0,Y 235.216,Z 316.184,A -85,B 0,C 180,E1 -19810.327,E2 -19810.327} C_VEL
LIN {X 0,Y 235.078,Z 316.201,A -85,B 0,C 180,E1 -19815.608,E2 -19815.608} C_VEL
LIN {X 0,Y 234.974,Z 316.215,A -85,B 0,C 180,E1 -19819.208,E2 -19819.208} C_VEL
LIN {X 0,Y 234.941,Z 316.219,A -85,B 0,C 180,E1 -19822.885,E2 -19822.885} C_VEL
LIN {X 0,Y 234.925,Z 316.22,A -85,B 0,C 180,E1 -19824.176,E2 -19824.176} C_VEL
LIN {X 0,Y 234.302,Z 316.304,A -85,B 0,C 180,E1 -19825.606,E2 -19825.606} C_VEL
LIN {X 0,Y 231.475,Z 316.663,A -85,B 0,C 180,E1 -19827.939,E2 -19827.939} C_VEL
LIN {X 0,Y 229.028,Z 316.965,A -85,B 0,C 180,E1 -19829.841,E2 -19829.841} C_VEL
LIN {X 0,Y 227.949,Z 317.093,A -85,B 0,C 180,E1 -19831.317,E2 -19831.317} C_VEL
LIN {X 0,Y 227.847,Z 317.102,A -85,B 0,C 180,E1 -19831.818,E2 -19831.818} C_VEL
LIN {X 0,Y 227.868,Z 317.101,A -85,B 0,C 180,E1 -19835.874,E2 -19835.874} C_VEL
LIN {X 0,Y 227.803,Z 317.108,A -85,B 0,C 180,E1 -19840.381,E2 -19840.381} C_VEL
LIN {X 0,Y 227.813,Z 317.109,A -85,B 0,C 180,E1 -19845.198,E2 -19845.198} C_VEL
LIN {X 0,Y 227.803,Z 317.102,A -85,B 0,C 180,E1 -19849.617,E2 -19849.617} C_VEL
LIN {X 0,Y 227.927,Z 317.241,A -85,B 0,C 180,E1 -19852.046,E2 -19852.046} C_VEL
LIN {X 0,Y 230.123,Z 326.647,A -85,B 0,C 180,E1 -19855.934,E2 -19855.934} C_VEL
LIN {X 0,Y 231.134,Z 331.305,A -85,B 0,C 180,E1 -19857.714,E2 -19857.714} C_VEL
LIN {X 0,Y 237.692,Z 348.612,A -85,B 0,C 180,E1 -19859.136,E2 -19859.136} C_VEL
LIN {X 0,Y 240.966,Z 375.412,A -85,B 0,C 180,E1 -19860.402,E2 -19860.402} C_VEL
LIN {X 0,Y 242.099,Z 387.123,A -85,B 0,C 180,E1 -19860.907,E2 -19860.907} C_VEL
LIN {X 0,Y 240.412,Z 440.082,A -85,B 0,C 180,E1 -19862.466,E2 -19862.466} C_VEL
LIN {X 0,Y 239.327,Z 453.454,A -85,B 0,C 180,E1 -19863.159,E2 -19863.159} C_VEL
LIN {X 0,Y 237.835,Z 466.255,A -85,B 0,C 180,E1 -19864.159,E2 -19864.159} C_VEL
LIN {X 0,Y 236.216,Z 477.624,A -85,B 0,C 180,E1 -19865.383,E2 -19865.383} C_VEL
LIN {X 0,Y 234.356,Z 488.034,A -85,B 0,C 180,E1 -19866.82,E2 -19866.82} C_VEL
LIN {X 0,Y 232.362,Z 498.811,A -85,B 0,C 180,E1 -19868.717,E2 -19868.717} C_VEL
LIN {X 0,Y 230.599,Z 508.522,A -85,B 0,C 180,E1 -19870.872,E2 -19870.872} C_VEL
LIN {X 0,Y 229.151,Z 516.482,A -85,B 0,C 180,E1 -19873.059,E2 -19873.059} C_VEL
LIN {X 0,Y 227.712,Z 524.224,A -85,B 0,C 180,E1 -19875.704,E2 -19875.704} C_VEL
LIN {X 0,Y 226.626,Z 530.435,A -85,B 0,C 180,E1 -19878.37,E2 -19878.37} C_VEL
LIN {X 0,Y 226.071,Z 535.366,A -85,B 0,C 180,E1 -19881.057,E2 -19881.057} C_VEL
LIN {X 0,Y 225.765,Z 539.143,A -85,B 0,C 180,E1 -19883.744,E2 -19883.744} C_VEL
LIN {X 0,Y 225.75,Z 541.881,A -85,B 0,C 180,E1 -19886.429,E2 -19886.429} C_VEL
LIN {X 0,Y 225.855,Z 543.166,A -85,B 0,C 180,E1 -19888.216,E2 -19888.216} C_VEL
LIN {X 0,Y 225.878,Z 544.043,A -85,B 0,C 180,E1 -19889.999,E2 -19889.999} C_VEL
LIN {X 0,Y 225.807,Z 544.478,A -85,B 0,C 180,E1 -19891.782,E2 -19891.782} C_VEL
LIN {X 0,Y 225.683,Z 544.139,A -85,B 0,C 180,E1 -19895.359,E2 -19895.359} C_VEL
LIN {X 0,Y 225.768,Z 543.394,A -85,B 0,C 180,E1 -19897.152,E2 -19897.152} C_VEL
LIN {X 0,Y 226.053,Z 542.241,A -85,B 0,C 180,E1 -19898.942,E2 -19898.942} C_VEL
LIN {X 0,Y 226.532,Z 540.656,A -85,B 0,C 180,E1 -19900.727,E2 -19900.727} C_VEL
LIN {X 0,Y 227.498,Z 537.502,A -85,B 0,C 180,E1 -19903.396,E2 -19903.396} C_VEL
LIN {X 0,Y 229.091,Z 533.315,A -85,B 0,C 180,E1 -19906.026,E2 -19906.026} C_VEL
LIN {X 0,Y 231.493,Z 526.964,A -85,B 0,C 180,E1 -19909.047,E2 -19909.047} C_VEL
LIN {X 0,Y 233.931,Z 520.078,A -85,B 0,C 180,E1 -19911.593,E2 -19911.593} C_VEL
LIN {X 0,Y 236.916,Z 511.508,A -85,B 0,C 180,E1 -19914.071,E2 -19914.071} C_VEL
LIN {X 0,Y 239.898,Z 502.735,A -85,B 0,C 180,E1 -19916.067,E2 -19916.067} C_VEL
LIN {X 0,Y 243.119,Z 491.964,A -85,B 0,C 180,E1 -19918.017,E2 -19918.017} C_VEL
LIN {X 0,Y 246.017,Z 481.191,A -85,B 0,C 180,E1 -19919.522,E2 -19919.522} C_VEL
LIN {X 0,Y 248.232,Z 471.112,A -85,B 0,C 180,E1 -19920.637,E2 -19920.637} C_VEL
LIN {X 0,Y 250.422,Z 459.139,A -85,B 0,C 180,E1 -19921.631,E2 -19921.631} C_VEL
LIN {X 0,Y 252.214,Z 445.898,A -85,B 0,C 180,E1 -19922.398,E2 -19922.398} C_VEL
LIN {X 0,Y 253.159,Z 432.955,A -85,B 0,C 180,E1 -19922.874,E2 -19922.874} C_VEL
LIN {X 0,Y 255.04,Z 391.459,A -85,B 0,C 180,E1 -19923.998,E2 -19923.998} C_VEL
LIN {X 0,Y 251.992,Z 370.16,A -85,B 0,C 180,E1 -19925.292,E2 -19925.292} C_VEL
LIN {X 0,Y 245.657,Z 355.801,A -85,B 0,C 180,E1 -19927.031,E2 -19927.031} C_VEL
LIN {X 0,Y 239.357,Z 343.443,A -85,B 0,C 180,E1 -19928.825,E2 -19928.825} C_VEL
LIN {X 0,Y 233.971,Z 333.825,A -85,B 0,C 180,E1 -19930.444,E2 -19930.444} C_VEL
LIN {X 0,Y 231.464,Z 329.299,A -85,B 0,C 180,E1 -19931.283,E2 -19931.283} C_VEL
LIN {X 0,Y 229.307,Z 321.887,A -85,B 0,C 180,E1 -19935.177,E2 -19935.177} C_VEL
LIN {X 0,Y 227.823,Z 317.105,A -85,B 0,C 180,E1 -19937.988,E2 -19937.988} C_VEL
LIN {X 0,Y 227.841,Z 317.096,A -85,B 0,C 180,E1 -19941.909,E2 -19941.909} C_VEL
LIN {X 0,Y 227.876,Z 317.095,A -85,B 0,C 180,E1 -19946.377,E2 -19946.377} C_VEL
LIN {X 0,Y 227.914,Z 317.093,A -85,B 0,C 180,E1 -19950.437,E2 -19950.437} C_VEL
LIN {X 0,Y 227.925,Z 317.089,A -85,B 0,C 180,E1 -19954.426,E2 -19954.426} C_VEL
LIN {X 0,Y 227.978,Z 317.084,A -85,B 0,C 180,E1 -19958.289,E2 -19958.289} C_VEL
LIN {X 0,Y 228.031,Z 317.073,A -85,B 0,C 180,E1 -19962.826,E2 -19962.826} C_VEL
LIN {X 0,Y 228.078,Z 317.075,A -85,B 0,C 180,E1 -19965.729,E2 -19965.729} C_VEL
LIN {X 0,Y 228.322,Z 317.037,A -85,B 0,C 180,E1 -19971.147,E2 -19971.147} C_VEL
LIN {X 0,Y 228.355,Z 317.033,A -85,B 0,C 180,E1 -19972.929,E2 -19972.929} C_VEL
LIN {X 0,Y 228.552,Z 317.014,A -85,B 0,C 180,E1 -19978.238,E2 -19978.238} C_VEL
LIN {X 0,Y 228.552,Z 317.01,A -85,B 0,C 180,E1 -19981.763,E2 -19981.763} C_VEL
LIN {X 0,Y 228.355,Z 317.04,A -85,B 0,C 180,E1 -19987.072,E2 -19987.072} C_VEL
LIN {X 0,Y 228.169,Z 317.059,A -85,B 0,C 180,E1 -19990.651,E2 -19990.651} C_VEL
LIN {X 0,Y 228.055,Z 317.076,A -85,B 0,C 180,E1 -19996.103,E2 -19996.103} C_VEL
LIN {X 0,Y 227.94,Z 317.091,A -85,B 0,C 180,E1 -19999.826,E2 -19999.826} C_VEL
LIN {X 0,Y 227.912,Z 317.095,A -85,B 0,C 180,E1 -20003.633,E2 -20003.633} C_VEL
LIN {X 0,Y 227.877,Z 317.098,A -85,B 0,C 180,E1 -20007.557,E2 -20007.557} C_VEL
LIN {X 0,Y 227.865,Z 317.094,A -85,B 0,C 180,E1 -20011.624,E2 -20011.624} C_VEL
LIN {X 0,Y 227.879,Z 317.091,A -85,B 0,C 180,E1 -20015.873,E2 -20015.873} C_VEL
LIN {X 0,Y 227.88,Z 317.112,A -85,B 0,C 180,E1 -20018.994,E2 -20018.994} C_VEL
LIN {X 0,Y 228.882,Z 319.947,A -85,B 0,C 180,E1 -20019.381,E2 -20019.381} C_VEL
LIN {X 0,Y 231.077,Z 322.489,A -85,B 0,C 180,E1 -20020.05,E2 -20020.05} C_VEL
LIN {X 0,Y 233.112,Z 325.729,A -85,B 0,C 180,E1 -20020.691,E2 -20020.691} C_VEL
LIN {X 0,Y 234.509,Z 327.633,A -85,B 0,C 180,E1 -20021.106,E2 -20021.106} C_VEL
LIN {X 0,Y 240.422,Z 336.561,A -85,B 0,C 180,E1 -20022.815,E2 -20022.815} C_VEL
LIN {X 0,Y 247.646,Z 348.284,A -85,B 0,C 180,E1 -20024.763,E2 -20024.763} C_VEL
LIN {X 0,Y 254.068,Z 361.041,A -85,B 0,C 180,E1 -20026.441,E2 -20026.441} C_VEL
LIN {X 0,Y 256.133,Z 365.666,A -85,B 0,C 180,E1 -20026.972,E2 -20026.972} C_VEL
LIN {X 0,Y 253.502,Z 420.071,A -85,B 0,C 180,E1 -20028.457,E2 -20028.457} C_VEL
LIN {X 0,Y 252.411,Z 433.059,A -85,B 0,C 180,E1 -20029.108,E2 -20029.108} C_VEL
LIN {X 0,Y 250.561,Z 446.386,A -85,B 0,C 180,E1 -20030.088,E2 -20030.088} C_VEL
LIN {X 0,Y 248.26,Z 457.832,A -85,B 0,C 180,E1 -20031.221,E2 -20031.221} C_VEL
LIN {X 0,Y 245.61,Z 469.625,A -85,B 0,C 180,E1 -20032.81,E2 -20032.81} C_VEL
LIN {X 0,Y 242.871,Z 480.184,A -85,B 0,C 180,E1 -20034.639,E2 -20034.639} C_VEL
LIN {X 0,Y 239.906,Z 489.589,A -85,B 0,C 180,E1 -20036.684,E2 -20036.684} C_VEL
LIN {X 0,Y 236.728,Z 498.794,A -85,B 0,C 180,E1 -20039.246,E2 -20039.246} C_VEL
LIN {X 0,Y 234.033,Z 505.908,A -85,B 0,C 180,E1 -20041.774,E2 -20041.774} C_VEL
LIN {X 0,Y 232.036,Z 510.766,A -85,B 0,C 180,E1 -20043.95,E2 -20043.95} C_VEL
LIN {X 0,Y 230.074,Z 515.45,A -85,B 0,C 180,E1 -20046.604,E2 -20046.604} C_VEL
LIN {X 0,Y 228.969,Z 517.924,A -85,B 0,C 180,E1 -20048.389,E2 -20048.389} C_VEL
LIN {X 0,Y 228.041,Z 519.916,A -85,B 0,C 180,E1 -20050.185,E2 -20050.185} C_VEL
LIN {X 0,Y 227.319,Z 521.483,A -85,B 0,C 180,E1 -20051.992,E2 -20051.992} C_VEL
LIN {X 0,Y 226.701,Z 522.688,A -85,B 0,C 180,E1 -20053.956,E2 -20053.956} C_VEL
LIN {X 0,Y 225.928,Z 523.622,A -85,B 0,C 180,E1 -20057.424,E2 -20057.424} C_VEL
LIN {X 0,Y 225.73,Z 523.541,A -85,B 0,C 180,E1 -20059.235,E2 -20059.235} C_VEL
LIN {X 0,Y 225.673,Z 523.047,A -85,B 0,C 180,E1 -20061.043,E2 -20061.043} C_VEL
LIN {X 0,Y 225.96,Z 520.98,A -85,B 0,C 180,E1 -20064.446,E2 -20064.446} C_VEL
LIN {X 0,Y 226.207,Z 518.075,A -85,B 0,C 180,E1 -20067.33,E2 -20067.33} C_VEL
LIN {X 0,Y 226.829,Z 514.316,A -85,B 0,C 180,E1 -20070.001,E2 -20070.001} C_VEL
LIN {X 0,Y 227.639,Z 509.454,A -85,B 0,C 180,E1 -20072.655,E2 -20072.655} C_VEL
LIN {X 0,Y 228.82,Z 503.333,A -85,B 0,C 180,E1 -20075.288,E2 -20075.288} C_VEL
LIN {X 0,Y 230.381,Z 495.719,A -85,B 0,C 180,E1 -20077.891,E2 -20077.891} C_VEL
LIN {X 0,Y 232.299,Z 486.153,A -85,B 0,C 180,E1 -20080.46,E2 -20080.46} C_VEL
LIN {X 0,Y 234.202,Z 476.286,A -85,B 0,C 180,E1 -20082.567,E2 -20082.567} C_VEL
LIN {X 0,Y 236.113,Z 465.162,A -85,B 0,C 180,E1 -20084.436,E2 -20084.436} C_VEL
LIN {X 0,Y 237.733,Z 454.274,A -85,B 0,C 180,E1 -20085.871,E2 -20085.871} C_VEL
LIN {X 0,Y 239.053,Z 442.286,A -85,B 0,C 180,E1 -20087.098,E2 -20087.098} C_VEL
LIN {X 0,Y 240.177,Z 429.879,A -85,B 0,C 180,E1 -20088.005,E2 -20088.005} C_VEL
LIN {X 0,Y 240.833,Z 417.054,A -85,B 0,C 180,E1 -20088.614,E2 -20088.614} C_VEL
LIN {X 0,Y 243.109,Z 351.229,A -85,B 0,C 180,E1 -20090.502,E2 -20090.502} C_VEL
LIN {X 0,Y 238.221,Z 338.521,A -85,B 0,C 180,E1 -20091.501,E2 -20091.501} C_VEL
LIN {X 0,Y 231.858,Z 325.463,A -85,B 0,C 180,E1 -20092.758,E2 -20092.758} C_VEL
LIN {X 0,Y 228.146,Z 318.271,A -85,B 0,C 180,E1 -20093.516,E2 -20093.516} C_VEL
LIN {X 0,Y 227.899,Z 317.087,A -85,B 0,C 180,E1 -20093.635,E2 -20093.635} C_VEL
LIN {X 0,Y 227.86,Z 317.097,A -85,B 0,C 180,E1 -20097.56,E2 -20097.56} C_VEL
LIN {X 0,Y 227.861,Z 317.101,A -85,B 0,C 180,E1 -20101.625,E2 -20101.625} C_VEL
LIN {X 0,Y 227.87,Z 317.099,A -85,B 0,C 180,E1 -20105.875,E2 -20105.875} C_VEL
LIN {X 0,Y 227.805,Z 317.101,A -85,B 0,C 180,E1 -20110.383,E2 -20110.383} C_VEL
LIN {X 0,Y 227.815,Z 317.105,A -85,B 0,C 180,E1 -20115.199,E2 -20115.199} C_VEL
LIN {X 0,Y 227.802,Z 317.104,A -85,B 0,C 180,E1 -20119.617,E2 -20119.617} C_VEL
LIN {X 0,Y 227.869,Z 317.089,A -85,B 0,C 180,E1 -20124.125,E2 -20124.125} C_VEL
LIN {X 0,Y 227.861,Z 317.099,A -85,B 0,C 180,E1 -20128.376,E2 -20128.376} C_VEL
LIN {X 0,Y 227.853,Z 317.095,A -85,B 0,C 180,E1 -20132.44,E2 -20132.44} C_VEL
LIN {X 0,Y 227.887,Z 317.089,A -85,B 0,C 180,E1 -20136.364,E2 -20136.364} C_VEL
LIN {X 0,Y 227.929,Z 317.092,A -85,B 0,C 180,E1 -20140.173,E2 -20140.173} C_VEL
LIN {X 0,Y 228.035,Z 317.061,A -85,B 0,C 180,E1 -20143.896,E2 -20143.896} C_VEL
LIN {X 0,Y 228.063,Z 317.068,A -85,B 0,C 180,E1 -20147.542,E2 -20147.542} C_VEL
LIN {X 0,Y 228.262,Z 317.048,A -85,B 0,C 180,E1 -20151.144,E2 -20151.144} C_VEL
LIN {X 0,Y 228.311,Z 317.036,A -85,B 0,C 180,E1 -20152.927,E2 -20152.927} C_VEL
LIN {X 0,Y 228.539,Z 317.009,A -85,B 0,C 180,E1 -20158.237,E2 -20158.237} C_VEL
LIN {X 0,Y 228.539,Z 317.016,A -85,B 0,C 180,E1 -20161.762,E2 -20161.762} C_VEL
LIN {X 0,Y 228.304,Z 317.029,A -85,B 0,C 180,E1 -20167.073,E2 -20167.073} C_VEL
LIN {X 0,Y 228.146,Z 317.067,A -85,B 0,C 180,E1 -20170.651,E2 -20170.651} C_VEL
LIN {X 0,Y 228.037,Z 317.076,A -85,B 0,C 180,E1 -20174.273,E2 -20174.273} C_VEL
LIN {X 0,Y 227.934,Z 317.09,A -85,B 0,C 180,E1 -20177.959,E2 -20177.959} C_VEL
LIN {X 0,Y 227.908,Z 317.096,A -85,B 0,C 180,E1 -20182.312,E2 -20182.312} C_VEL
LIN {X 0,Y 227.925,Z 317.094,A -85,B 0,C 180,E1 -20186.591,E2 -20186.591} C_VEL
LIN {X 0,Y 227.873,Z 317.1,A -85,B 0,C 180,E1 -20190.278,E2 -20190.278} C_VEL
LIN {X 0,Y 227.847,Z 317.102,A -85,B 0,C 180,E1 -20191.818,E2 -20191.818} C_VEL
LIN {X 0,Y 227.148,Z 317.193,A -85,B 0,C 180,E1 -20193.293,E2 -20193.293} C_VEL
LIN {X 0,Y 224.309,Z 317.545,A -85,B 0,C 180,E1 -20195.702,E2 -20195.702} C_VEL
LIN {X 0,Y 221.91,Z 317.847,A -85,B 0,C 180,E1 -20197.666,E2 -20197.666} C_VEL
LIN {X 0,Y 220.87,Z 317.975,A -85,B 0,C 180,E1 -20199.19,E2 -20199.19} C_VEL
LIN {X 0,Y 220.779,Z 317.984,A -85,B 0,C 180,E1 -20199.707,E2 -20199.707} C_VEL
LIN {X 0,Y 220.756,Z 317.986,A -85,B 0,C 180,E1 -20204.458,E2 -20204.458} C_VEL
LIN {X 0,Y 220.75,Z 317.986,A -85,B 0,C 180,E1 -20208.041,E2 -20208.041} C_VEL
LIN {X 0,Y 220.852,Z 318.132,A -85,B 0,C 180,E1 -20211.314,E2 -20211.314} C_VEL
LIN {X 0,Y 223.187,Z 327.782,A -85,B 0,C 180,E1 -20215.471,E2 -20215.471} C_VEL
LIN {X 0,Y 223.779,Z 330.724,A -85,B 0,C 180,E1 -20216.674,E2 -20216.674} C_VEL
LIN {X 0,Y 231.438,Z 350.397,A -85,B 0,C 180,E1 -20218.413,E2 -20218.413} C_VEL
LIN {X 0,Y 234.3,Z 373.706,A -85,B 0,C 180,E1 -20219.563,E2 -20219.563} C_VEL
LIN {X 0,Y 235.652,Z 388.329,A -85,B 0,C 180,E1 -20220.214,E2 -20220.214} C_VEL
LIN {X 0,Y 233.877,Z 440.777,A -85,B 0,C 180,E1 -20221.812,E2 -20221.812} C_VEL
LIN {X 0,Y 232.667,Z 454.574,A -85,B 0,C 180,E1 -20222.57,E2 -20222.57} C_VEL
LIN {X 0,Y 231.142,Z 466.957,A -85,B 0,C 180,E1 -20223.596,E2 -20223.596} C_VEL
LIN {X 0,Y 229.193,Z 479.648,A -85,B 0,C 180,E1 -20225.061,E2 -20225.061} C_VEL
LIN {X 0,Y 227.185,Z 490.953,A -85,B 0,C 180,E1 -20226.769,E2 -20226.769} C_VEL
LIN {X 0,Y 225.123,Z 501.1,A -85,B 0,C 180,E1 -20228.72,E2 -20228.72} C_VEL
LIN {X 0,Y 223.149,Z 510.741,A -85,B 0,C 180,E1 -20231.061,E2 -20231.061} C_VEL
LIN {X 0,Y 222.351,Z 515.769,A -85,B 0,C 180,E1 -20232.525,E2 -20232.525} C_VEL
LIN {X 0,Y 220.79,Z 523.602,A -85,B 0,C 180,E1 -20235.246,E2 -20235.246} C_VEL
LIN {X 0,Y 219.633,Z 529.869,A -85,B 0,C 180,E1 -20237.994,E2 -20237.994} C_VEL
LIN {X 0,Y 219.023,Z 534.849,A -85,B 0,C 180,E1 -20240.766,E2 -20240.766} C_VEL
LIN {X 0,Y 218.7,Z 538.675,A -85,B 0,C 180,E1 -20243.541,E2 -20243.541} C_VEL
LIN {X 0,Y 218.658,Z 541.456,A -85,B 0,C 180,E1 -20246.313,E2 -20246.313} C_VEL
LIN {X 0,Y 218.761,Z 542.763,A -85,B 0,C 180,E1 -20248.158,E2 -20248.158} C_VEL
LIN {X 0,Y 218.808,Z 543.662,A -85,B 0,C 180,E1 -20249.999,E2 -20249.999} C_VEL
LIN {X 0,Y 218.713,Z 544.136,A -85,B 0,C 180,E1 -20251.84,E2 -20251.84} C_VEL
LIN {X 0,Y 218.586,Z 543.837,A -85,B 0,C 180,E1 -20255.534,E2 -20255.534} C_VEL
LIN {X 0,Y 219.018,Z 541.999,A -85,B 0,C 180,E1 -20259.231,E2 -20259.231} C_VEL
LIN {X 0,Y 219.526,Z 540.44,A -85,B 0,C 180,E1 -20261.073,E2 -20261.073} C_VEL
LIN {X 0,Y 220.567,Z 537.333,A -85,B 0,C 180,E1 -20263.825,E2 -20263.825} C_VEL
LIN {X 0,Y 222.265,Z 533.196,A -85,B 0,C 180,E1 -20266.533,E2 -20266.533} C_VEL
LIN {X 0,Y 224.791,Z 526.898,A -85,B 0,C 180,E1 -20269.638,E2 -20269.638} C_VEL
LIN {X 0,Y 227.329,Z 520.072,A -85,B 0,C 180,E1 -20272.253,E2 -20272.253} C_VEL
LIN {X 0,Y 230.453,Z 511.606,A -85,B 0,C 180,E1 -20274.791,E2 -20274.791} C_VEL
LIN {X 0,Y 233.554,Z 502.918,A -85,B 0,C 180,E1 -20276.831,E2 -20276.831} C_VEL
LIN {X 0,Y 236.881,Z 492.251,A -85,B 0,C 180,E1 -20278.823,E2 -20278.823} C_VEL
LIN {X 0,Y 239.877,Z 481.656,A -85,B 0,C 180,E1 -20280.356,E2 -20280.356} C_VEL
LIN {X 0,Y 242.601,Z 469.845,A -85,B 0,C 180,E1 -20281.672,E2 -20281.672} C_VEL
LIN {X 0,Y 244.876,Z 457.585,A -85,B 0,C 180,E1 -20282.677,E2 -20282.677} C_VEL
LIN {X 0,Y 246.594,Z 444.702,A -85,B 0,C 180,E1 -20283.418,E2 -20283.418} C_VEL
LIN {X 0,Y 247.584,Z 430.91,A -85,B 0,C 180,E1 -20283.901,E2 -20283.901} C_VEL
LIN {X 0,Y 249.343,Z 391.66,A -85,B 0,C 180,E1 -20285,E2 -20285} C_VEL
LIN {X 0,Y 246.573,Z 372.646,A -85,B 0,C 180,E1 -20286.218,E2 -20286.218} C_VEL
LIN {X 0,Y 239.521,Z 356.86,A -85,B 0,C 180,E1 -20288.257,E2 -20288.257} C_VEL
LIN {X 0,Y 232.88,Z 343.991,A -85,B 0,C 180,E1 -20290.274,E2 -20290.274} C_VEL
LIN {X 0,Y 228.828,Z 337.092,A -85,B 0,C 180,E1 -20291.56,E2 -20291.56} C_VEL
LIN {X 0,Y 226.716,Z 333.476,A -85,B 0,C 180,E1 -20292.26,E2 -20292.26} C_VEL
LIN {X 0,Y 224.317,Z 329.413,A -85,B 0,C 180,E1 -20293.082,E2 -20293.082} C_VEL
LIN {X 0,Y 224.09,Z 328.861,A -85,B 0,C 180,E1 -20293.184,E2 -20293.184} C_VEL
LIN {X 0,Y 221.786,Z 321.509,A -85,B 0,C 180,E1 -20297.392,E2 -20297.392} C_VEL
LIN {X 0,Y 220.794,Z 317.976,A -85,B 0,C 180,E1 -20299.612,E2 -20299.612} C_VEL
LIN {X 0,Y 220.821,Z 317.972,A -85,B 0,C 180,E1 -20302.792,E2 -20302.792} C_VEL
LIN {X 0,Y 220.814,Z 317.976,A -85,B 0,C 180,E1 -20307.244,E2 -20307.244} C_VEL
LIN {X 0,Y 220.832,Z 317.967,A -85,B 0,C 180,E1 -20311.486,E2 -20311.486} C_VEL
LIN {X 0,Y 220.867,Z 317.961,A -85,B 0,C 180,E1 -20315.565,E2 -20315.565} C_VEL
LIN {X 0,Y 220.896,Z 317.958,A -85,B 0,C 180,E1 -20319.515,E2 -20319.515} C_VEL
LIN {X 0,Y 221.013,Z 317.945,A -85,B 0,C 180,E1 -20323.37,E2 -20323.37} C_VEL
LIN {X 0,Y 221.109,Z 317.938,A -85,B 0,C 180,E1 -20329.006,E2 -20329.006} C_VEL
LIN {X 0,Y 221.292,Z 317.911,A -85,B 0,C 180,E1 -20332.702,E2 -20332.702} C_VEL
LIN {X 0,Y 221.51,Z 317.891,A -85,B 0,C 180,E1 -20338.182,E2 -20338.182} C_VEL
LIN {X 0,Y 221.51,Z 317.888,A -85,B 0,C 180,E1 -20341.819,E2 -20341.819} C_VEL
LIN {X 0,Y 221.308,Z 317.917,A -85,B 0,C 180,E1 -20347.298,E2 -20347.298} C_VEL
LIN {X 0,Y 221.114,Z 317.94,A -85,B 0,C 180,E1 -20350.995,E2 -20350.995} C_VEL
LIN {X 0,Y 221.014,Z 317.948,A -85,B 0,C 180,E1 -20356.631,E2 -20356.631} C_VEL
LIN {X 0,Y 220.89,Z 317.965,A -85,B 0,C 180,E1 -20360.487,E2 -20360.487} C_VEL
LIN {X 0,Y 220.865,Z 317.968,A -85,B 0,C 180,E1 -20364.436,E2 -20364.436} C_VEL
LIN {X 0,Y 220.825,Z 317.97,A -85,B 0,C 180,E1 -20368.516,E2 -20368.516} C_VEL
LIN {X 0,Y 220.815,Z 317.97,A -85,B 0,C 180,E1 -20372.757,E2 -20372.757} C_VEL
LIN {X 0,Y 220.834,Z 317.975,A -85,B 0,C 180,E1 -20377.074,E2 -20377.074} C_VEL
LIN {X 0,Y 221.705,Z 320.607,A -85,B 0,C 180,E1 -20377.463,E2 -20377.463} C_VEL
LIN {X 0,Y 223.577,Z 322.771,A -85,B 0,C 180,E1 -20378.091,E2 -20378.091} C_VEL
LIN {X 0,Y 224.378,Z 323.798,A -85,B 0,C 180,E1 -20378.359,E2 -20378.359} C_VEL
LIN {X 0,Y 226.571,Z 327.029,A -85,B 0,C 180,E1 -20379.094,E2 -20379.094} C_VEL
LIN {X 0,Y 228.114,Z 329.334,A -85,B 0,C 180,E1 -20379.599,E2 -20379.599} C_VEL
LIN {X 0,Y 232.928,Z 336.149,A -85,B 0,C 180,E1 -20381.089,E2 -20381.089} C_VEL
LIN {X 0,Y 241.655,Z 350.197,A -85,B 0,C 180,E1 -20383.616,E2 -20383.616} C_VEL
LIN {X 0,Y 246.445,Z 359.181,A -85,B 0,C 180,E1 -20384.935,E2 -20384.935} C_VEL
LIN {X 0,Y 250.475,Z 367.844,A -85,B 0,C 180,E1 -20386.027,E2 -20386.027} C_VEL
LIN {X 0,Y 247.826,Z 420.428,A -85,B 0,C 180,E1 -20387.487,E2 -20387.487} C_VEL
LIN {X 0,Y 246.637,Z 433.82,A -85,B 0,C 180,E1 -20388.176,E2 -20388.176} C_VEL
LIN {X 0,Y 244.655,Z 447.315,A -85,B 0,C 180,E1 -20389.194,E2 -20389.194} C_VEL
LIN {X 0,Y 242.283,Z 458.591,A -85,B 0,C 180,E1 -20390.346,E2 -20390.346} C_VEL
LIN {X 0,Y 239.517,Z 470.304,A -85,B 0,C 180,E1 -20391.963,E2 -20391.963} C_VEL
LIN {X 0,Y 236.661,Z 480.799,A -85,B 0,C 180,E1 -20393.829,E2 -20393.829} C_VEL
LIN {X 0,Y 233.869,Z 489.311,A -85,B 0,C 180,E1 -20395.706,E2 -20395.706} C_VEL
LIN {X 0,Y 230.535,Z 498.483,A -85,B 0,C 180,E1 -20398.274,E2 -20398.274} C_VEL
LIN {X 0,Y 227.663,Z 505.831,A -85,B 0,C 180,E1 -20400.91,E2 -20400.91} C_VEL
LIN {X 0,Y 225.513,Z 510.763,A -85,B 0,C 180,E1 -20403.137,E2 -20403.137} C_VEL
LIN {X 0,Y 223.417,Z 515.52,A -85,B 0,C 180,E1 -20405.863,E2 -20405.863} C_VEL
LIN {X 0,Y 221.722,Z 519.125,A -85,B 0,C 180,E1 -20408.623,E2 -20408.623} C_VEL
LIN {X 0,Y 220.434,Z 521.684,A -85,B 0,C 180,E1 -20411.409,E2 -20411.409} C_VEL
LIN {X 0,Y 219.679,Z 523.057,A -85,B 0,C 180,E1 -20413.695,E2 -20413.695} C_VEL
LIN {X 0,Y 218.891,Z 523.942,A -85,B 0,C 180,E1 -20417.013,E2 -20417.013} C_VEL
LIN {X 0,Y 218.598,Z 523.446,A -85,B 0,C 180,E1 -20420.751,E2 -20420.751} C_VEL
LIN {X 0,Y 218.646,Z 522.565,A -85,B 0,C 180,E1 -20422.614,E2 -20422.614} C_VEL
LIN {X 0,Y 218.889,Z 521.28,A -85,B 0,C 180,E1 -20424.474,E2 -20424.474} C_VEL
LIN {X 0,Y 219.119,Z 518.601,A -85,B 0,C 180,E1 -20427.244,E2 -20427.244} C_VEL
LIN {X 0,Y 219.712,Z 514.91,A -85,B 0,C 180,E1 -20430.001,E2 -20430.001} C_VEL
LIN {X 0,Y 220.575,Z 510.115,A -85,B 0,C 180,E1 -20432.741,E2 -20432.741} C_VEL
LIN {X 0,Y 221.767,Z 504.072,A -85,B 0,C 180,E1 -20435.457,E2 -20435.457} C_VEL
LIN {X 0,Y 223.371,Z 496.56,A -85,B 0,C 180,E1 -20438.141,E2 -20438.141} C_VEL
LIN {X 0,Y 225.014,Z 488.882,A -85,B 0,C 180,E1 -20440.347,E2 -20440.347} C_VEL
LIN {X 0,Y 227.089,Z 478.46,A -85,B 0,C 180,E1 -20442.74,E2 -20442.74} C_VEL
LIN {X 0,Y 229.056,Z 467.846,A -85,B 0,C 180,E1 -20444.664,E2 -20444.664} C_VEL
LIN {X 0,Y 230.749,Z 457.578,A -85,B 0,C 180,E1 -20446.137,E2 -20446.137} C_VEL
LIN {X 0,Y 232.21,Z 445.378,A -85,B 0,C 180,E1 -20447.505,E2 -20447.505} C_VEL
LIN {X 0,Y 233.504,Z 432.511,A -85,B 0,C 180,E1 -20448.538,E2 -20448.538} C_VEL
LIN {X 0,Y 234.259,Z 420.108,A -85,B 0,C 180,E1 -20449.214,E2 -20449.214} C_VEL
LIN {X 0,Y 236.789,Z 353.668,A -85,B 0,C 180,E1 -20451.171,E2 -20451.171} C_VEL
LIN {X 0,Y 234.105,Z 345.758,A -85,B 0,C 180,E1 -20451.771,E2 -20451.771} C_VEL
LIN {X 0,Y 227.512,Z 331.49,A -85,B 0,C 180,E1 -20453.136,E2 -20453.136} C_VEL
LIN {X 0,Y 221.036,Z 318.952,A -85,B 0,C 180,E1 -20454.516,E2 -20454.516} C_VEL
LIN {X 0,Y 220.843,Z 317.959,A -85,B 0,C 180,E1 -20454.627,E2 -20454.627} C_VEL
LIN {X 0,Y 220.809,Z 317.976,A -85,B 0,C 180,E1 -20458.519,E2 -20458.519} C_VEL
LIN {X 0,Y 220.817,Z 317.979,A -85,B 0,C 180,E1 -20462.757,E2 -20462.757} C_VEL
LIN {X 0,Y 220.807,Z 317.98,A -85,B 0,C 180,E1 -20467.276,E2 -20467.276} C_VEL
LIN {X 0,Y 220.753,Z 317.98,A -85,B 0,C 180,E1 -20471.958,E2 -20471.958} C_VEL
LIN {X 0,Y 220.757,Z 317.98,A -85,B 0,C 180,E1 -20475.541,E2 -20475.541} C_VEL
LIN {X 0,Y 220.785,Z 317.98,A -85,B 0,C 180,E1 -20480.458,E2 -20480.458} C_VEL
LIN {X 0,Y 220.83,Z 317.974,A -85,B 0,C 180,E1 -20482.793,E2 -20482.793} C_VEL
LIN {X 0,Y 220.817,Z 317.969,A -85,B 0,C 180,E1 -20487.243,E2 -20487.243} C_VEL
LIN {X 0,Y 220.806,Z 317.978,A -85,B 0,C 180,E1 -20491.481,E2 -20491.481} C_VEL
LIN {X 0,Y 220.838,Z 317.957,A -85,B 0,C 180,E1 -20495.561,E2 -20495.561} C_VEL
LIN {X 0,Y 220.883,Z 317.971,A -85,B 0,C 180,E1 -20499.512,E2 -20499.512} C_VEL
LIN {X 0,Y 220.996,Z 317.942,A -85,B 0,C 180,E1 -20503.368,E2 -20503.368} C_VEL
LIN {X 0,Y 221.068,Z 317.945,A -85,B 0,C 180,E1 -20509.003,E2 -20509.003} C_VEL
LIN {X 0,Y 221.248,Z 317.916,A -85,B 0,C 180,E1 -20512.7,E2 -20512.7} C_VEL
LIN {X 0,Y 221.472,Z 317.888,A -85,B 0,C 180,E1 -20518.181,E2 -20518.181} C_VEL
LIN {X 0,Y 221.473,Z 317.896,A -85,B 0,C 180,E1 -20521.818,E2 -20521.818} C_VEL
LIN {X 0,Y 221.242,Z 317.909,A -85,B 0,C 180,E1 -20527.3,E2 -20527.3} C_VEL
LIN {X 0,Y 221.066,Z 317.948,A -85,B 0,C 180,E1 -20530.996,E2 -20530.996} C_VEL
LIN {X 0,Y 220.982,Z 317.96,A -85,B 0,C 180,E1 -20536.632,E2 -20536.632} C_VEL
LIN {X 0,Y 220.858,Z 317.975,A -85,B 0,C 180,E1 -20540.489,E2 -20540.489} C_VEL
LIN {X 0,Y 220.849,Z 317.975,A -85,B 0,C 180,E1 -20544.437,E2 -20544.437} C_VEL
LIN {X 0,Y 220.804,Z 317.981,A -85,B 0,C 180,E1 -20548.518,E2 -20548.518} C_VEL
LIN {X 0,Y 220.814,Z 317.982,A -85,B 0,C 180,E1 -20552.756,E2 -20552.756} C_VEL
LIN {X 0,Y 220.805,Z 317.983,A -85,B 0,C 180,E1 -20557.274,E2 -20557.274} C_VEL
LIN {X 0,Y 220.779,Z 317.984,A -85,B 0,C 180,E1 -20559.707,E2 -20559.707} C_VEL
LIN {X 0,Y 220.081,Z 318.073,A -85,B 0,C 180,E1 -20561.227,E2 -20561.227} C_VEL
LIN {X 0,Y 217.189,Z 318.432,A -85,B 0,C 180,E1 -20563.707,E2 -20563.707} C_VEL
LIN {X 0,Y 214.753,Z 318.733,A -85,B 0,C 180,E1 -20565.732,E2 -20565.732} C_VEL
LIN {X 0,Y 213.726,Z 318.863,A -85,B 0,C 180,E1 -20567.306,E2 -20567.306} C_VEL
LIN {X 0,Y 213.651,Z 318.86,A -85,B 0,C 180,E1 -20567.84,E2 -20567.84} C_VEL
LIN {X 0,Y 213.755,Z 318.971,A -85,B 0,C 180,E1 -20570.504,E2 -20570.504} C_VEL
LIN {X 0,Y 215.931,Z 327.733,A -85,B 0,C 180,E1 -20574.457,E2 -20574.457} C_VEL
LIN {X 0,Y 216.571,Z 330.615,A -85,B 0,C 180,E1 -20575.606,E2 -20575.606} C_VEL
LIN {X 0,Y 222.672,Z 345.575,A -85,B 0,C 180,E1 -20577.06,E2 -20577.06} C_VEL
LIN {X 0,Y 225.541,Z 353.731,A -85,B 0,C 180,E1 -20577.749,E2 -20577.749} C_VEL
LIN {X 0,Y 228.571,Z 380.576,A -85,B 0,C 180,E1 -20579.088,E2 -20579.088} C_VEL
LIN {X 0,Y 229.261,Z 388.358,A -85,B 0,C 180,E1 -20579.444,E2 -20579.444} C_VEL
LIN {X 0,Y 227.447,Z 440.311,A -85,B 0,C 180,E1 -20581.067,E2 -20581.067} C_VEL
LIN {X 0,Y 226.206,Z 454.156,A -85,B 0,C 180,E1 -20581.844,E2 -20581.844} C_VEL
LIN {X 0,Y 224.623,Z 466.568,A -85,B 0,C 180,E1 -20582.893,E2 -20582.893} C_VEL
LIN {X 0,Y 222.767,Z 478.479,A -85,B 0,C 180,E1 -20584.29,E2 -20584.29} C_VEL
LIN {X 0,Y 220.787,Z 488.612,A -85,B 0,C 180,E1 -20585.804,E2 -20585.804} C_VEL
LIN {X 0,Y 218.654,Z 499.177,A -85,B 0,C 180,E1 -20587.809,E2 -20587.809} C_VEL
LIN {X 0,Y 216.579,Z 509.394,A -85,B 0,C 180,E1 -20590.288,E2 -20590.288} C_VEL
LIN {X 0,Y 215.201,Z 516.49,A -85,B 0,C 180,E1 -20592.416,E2 -20592.416} C_VEL
LIN {X 0,Y 213.645,Z 524.103,A -85,B 0,C 180,E1 -20595.229,E2 -20595.229} C_VEL
LIN {X 0,Y 212.368,Z 531.13,A -85,B 0,C 180,E1 -20598.546,E2 -20598.546} C_VEL
LIN {X 0,Y 211.83,Z 535.767,A -85,B 0,C 180,E1 -20601.413,E2 -20601.413} C_VEL
LIN {X 0,Y 211.573,Z 539.278,A -85,B 0,C 180,E1 -20604.28,E2 -20604.28} C_VEL
LIN {X 0,Y 211.571,Z 541.031,A -85,B 0,C 180,E1 -20606.189,E2 -20606.189} C_VEL
LIN {X 0,Y 211.67,Z 542.359,A -85,B 0,C 180,E1 -20608.096,E2 -20608.096} C_VEL
LIN {X 0,Y 211.74,Z 543.281,A -85,B 0,C 180,E1 -20609.999,E2 -20609.999} C_VEL
LIN {X 0,Y 211.622,Z 543.788,A -85,B 0,C 180,E1 -20611.902,E2 -20611.902} C_VEL
LIN {X 0,Y 211.512,Z 543.778,A -85,B 0,C 180,E1 -20614.572,E2 -20614.572} C_VEL
LIN {X 0,Y 211.631,Z 542.834,A -85,B 0,C 180,E1 -20617.632,E2 -20617.632} C_VEL
LIN {X 0,Y 211.999,Z 541.749,A -85,B 0,C 180,E1 -20619.54,E2 -20619.54} C_VEL
LIN {X 0,Y 212.513,Z 540.225,A -85,B 0,C 180,E1 -20621.444,E2 -20621.444} C_VEL
LIN {X 0,Y 213.66,Z 537.165,A -85,B 0,C 180,E1 -20624.281,E2 -20624.281} C_VEL
LIN {X 0,Y 215.459,Z 533.077,A -85,B 0,C 180,E1 -20627.07,E2 -20627.07} C_VEL
LIN {X 0,Y 218.094,Z 526.832,A -85,B 0,C 180,E1 -20630.267,E2 -20630.267} C_VEL
LIN {X 0,Y 220.743,Z 520.065,A -85,B 0,C 180,E1 -20632.954,E2 -20632.954} C_VEL
LIN {X 0,Y 224.038,Z 511.696,A -85,B 0,C 180,E1 -20635.551,E2 -20635.551} C_VEL
LIN {X 0,Y 227.249,Z 503.101,A -85,B 0,C 180,E1 -20637.638,E2 -20637.638} C_VEL
LIN {X 0,Y 230.704,Z 492.538,A -85,B 0,C 180,E1 -20639.67,E2 -20639.67} C_VEL
LIN {X 0,Y 233.808,Z 482.079,A -85,B 0,C 180,E1 -20641.231,E2 -20641.231} C_VEL
LIN {X 0,Y 236.602,Z 470.568,A -85,B 0,C 180,E1 -20642.572,E2 -20642.572} C_VEL
LIN {X 0,Y 238.957,Z 458.637,A -85,B 0,C 180,E1 -20643.592,E2 -20643.592} C_VEL
LIN {X 0,Y 240.888,Z 445.137,A -85,B 0,C 180,E1 -20644.4,E2 -20644.4} C_VEL
LIN {X 0,Y 241.891,Z 432.223,A -85,B 0,C 180,E1 -20644.89,E2 -20644.89} C_VEL
LIN {X 0,Y 243.791,Z 392.774,A -85,B 0,C 180,E1 -20646.004,E2 -20646.004} C_VEL
LIN {X 0,Y 241.403,Z 375.692,A -85,B 0,C 180,E1 -20647.129,E2 -20647.129} C_VEL
LIN {X 0,Y 234.528,Z 360.194,A -85,B 0,C 180,E1 -20649.22,E2 -20649.22} C_VEL
LIN {X 0,Y 228.455,Z 348.327,A -85,B 0,C 180,E1 -20651.162,E2 -20651.162} C_VEL
LIN {X 0,Y 223.068,Z 338.86,A -85,B 0,C 180,E1 -20652.986,E2 -20652.986} C_VEL
LIN {X 0,Y 219.46,Z 333.086,A -85,B 0,C 180,E1 -20654.268,E2 -20654.268} C_VEL
LIN {X 0,Y 216.629,Z 328.28,A -85,B 0,C 180,E1 -20655.385,E2 -20655.385} C_VEL
LIN {X 0,Y 214.735,Z 322.241,A -85,B 0,C 180,E1 -20659.113,E2 -20659.113} C_VEL
LIN {X 0,Y 213.718,Z 318.857,A -85,B 0,C 180,E1 -20661.449,E2 -20661.449} C_VEL
LIN {X 0,Y 213.753,Z 318.851,A -85,B 0,C 180,E1 -20666.018,E2 -20666.018} C_VEL
LIN {X 0,Y 213.777,Z 318.854,A -85,B 0,C 180,E1 -20670.454,E2 -20670.454} C_VEL
LIN {X 0,Y 213.8,Z 318.846,A -85,B 0,C 180,E1 -20674.702,E2 -20674.702} C_VEL
LIN {X 0,Y 213.829,Z 318.841,A -85,B 0,C 180,E1 -20678.805,E2 -20678.805} C_VEL
LIN {X 0,Y 213.94,Z 318.828,A -85,B 0,C 180,E1 -20682.804,E2 -20682.804} C_VEL
LIN {X 0,Y 213.976,Z 318.826,A -85,B 0,C 180,E1 -20686.708,E2 -20686.708} C_VEL
LIN {X 0,Y 214.193,Z 318.802,A -85,B 0,C 180,E1 -20690.558,E2 -20690.558} C_VEL
LIN {X 0,Y 214.109,Z 318.815,A -85,B 0,C 180,E1 -20694.349,E2 -20694.349} C_VEL
LIN {X 0,Y 214.443,Z 318.772,A -85,B 0,C 180,E1 -20698.122,E2 -20698.122} C_VEL
LIN {X 0,Y 214.548,Z 318.751,A -85,B 0,C 180,E1 -20700,E2 -20700} C_VEL
LIN {X 0,Y 214.443,Z 318.768,A -85,B 0,C 180,E1 -20701.879,E2 -20701.879} C_VEL
LIN {X 0,Y 214.245,Z 318.795,A -85,B 0,C 180,E1 -20707.54,E2 -20707.54} C_VEL
LIN {X 0,Y 214.045,Z 318.822,A -85,B 0,C 180,E1 -20711.362,E2 -20711.362} C_VEL
LIN {X 0,Y 213.932,Z 318.836,A -85,B 0,C 180,E1 -20715.238,E2 -20715.238} C_VEL
LIN {X 0,Y 213.866,Z 318.844,A -85,B 0,C 180,E1 -20719.185,E2 -20719.185} C_VEL
LIN {X 0,Y 213.845,Z 318.848,A -85,B 0,C 180,E1 -20723.228,E2 -20723.228} C_VEL
LIN {X 0,Y 213.827,Z 318.849,A -85,B 0,C 180,E1 -20727.451,E2 -20727.451} C_VEL
LIN {X 0,Y 213.766,Z 318.849,A -85,B 0,C 180,E1 -20731.739,E2 -20731.739} C_VEL
LIN {X 0,Y 213.768,Z 318.849,A -85,B 0,C 180,E1 -20734.941,E2 -20734.941} C_VEL
LIN {X 0,Y 214.681,Z 321.565,A -85,B 0,C 180,E1 -20735.393,E2 -20735.393} C_VEL
LIN {X 0,Y 216.699,Z 323.739,A -85,B 0,C 180,E1 -20736.133,E2 -20736.133} C_VEL
LIN {X 0,Y 217.558,Z 324.896,A -85,B 0,C 180,E1 -20736.452,E2 -20736.452} C_VEL
LIN {X 0,Y 219.501,Z 327.827,A -85,B 0,C 180,E1 -20737.172,E2 -20737.172} C_VEL
LIN {X 0,Y 220.843,Z 329.395,A -85,B 0,C 180,E1 -20737.635,E2 -20737.635} C_VEL
LIN {X 0,Y 229.183,Z 341.642,A -85,B 0,C 180,E1 -20740.41,E2 -20740.41} C_VEL
LIN {X 0,Y 237.021,Z 354.365,A -85,B 0,C 180,E1 -20742.782,E2 -20742.782} C_VEL
LIN {X 0,Y 241.801,Z 363.416,A -85,B 0,C 180,E1 -20744.16,E2 -20744.16} C_VEL
LIN {X 0,Y 244.916,Z 370.198,A -85,B 0,C 180,E1 -20745.048,E2 -20745.048} C_VEL
LIN {X 0,Y 242.243,Z 420.847,A -85,B 0,C 180,E1 -20746.476,E2 -20746.476} C_VEL
LIN {X 0,Y 240.979,Z 434.331,A -85,B 0,C 180,E1 -20747.183,E2 -20747.183} C_VEL
LIN {X 0,Y 239.031,Z 447.145,A -85,B 0,C 180,E1 -20748.161,E2 -20748.161} C_VEL
LIN {X 0,Y 236.376,Z 459.366,A -85,B 0,C 180,E1 -20749.43,E2 -20749.43} C_VEL
LIN {X 0,Y 233.564,Z 470.702,A -85,B 0,C 180,E1 -20751.028,E2 -20751.028} C_VEL
LIN {X 0,Y 230.521,Z 481.411,A -85,B 0,C 180,E1 -20752.979,E2 -20752.979} C_VEL
LIN {X 0,Y 227.286,Z 490.69,A -85,B 0,C 180,E1 -20755.108,E2 -20755.108} C_VEL
LIN {X 0,Y 223.859,Z 499.682,A -85,B 0,C 180,E1 -20757.745,E2 -20757.745} C_VEL
LIN {X 0,Y 220.871,Z 506.852,A -85,B 0,C 180,E1 -20760.45,E2 -20760.45} C_VEL
LIN {X 0,Y 218.235,Z 512.517,A -85,B 0,C 180,E1 -20763.203,E2 -20763.203} C_VEL
LIN {X 0,Y 216.056,Z 517.07,A -85,B 0,C 180,E1 -20766.115,E2 -20766.115} C_VEL
LIN {X 0,Y 214.432,Z 520.256,A -85,B 0,C 180,E1 -20768.869,E2 -20768.869} C_VEL
LIN {X 0,Y 213.562,Z 521.885,A -85,B 0,C 180,E1 -20770.788,E2 -20770.788} C_VEL
LIN {X 0,Y 212.663,Z 523.426,A -85,B 0,C 180,E1 -20773.414,E2 -20773.414} C_VEL
LIN {X 0,Y 211.874,Z 524.262,A -85,B 0,C 180,E1 -20776.575,E2 -20776.575} C_VEL
LIN {X 0,Y 211.507,Z 523.829,A -85,B 0,C 180,E1 -20780.438,E2 -20780.438} C_VEL
LIN {X 0,Y 211.554,Z 523.001,A -85,B 0,C 180,E1 -20782.365,E2 -20782.365} C_VEL
LIN {X 0,Y 211.802,Z 521.548,A -85,B 0,C 180,E1 -20784.545,E2 -20784.545} C_VEL
LIN {X 0,Y 212.139,Z 518.058,A -85,B 0,C 180,E1 -20788.103,E2 -20788.103} C_VEL
LIN {X 0,Y 212.87,Z 514.076,A -85,B 0,C 180,E1 -20790.947,E2 -20790.947} C_VEL
LIN {X 0,Y 214.043,Z 507.96,A -85,B 0,C 180,E1 -20794.238,E2 -20794.238} C_VEL
LIN {X 0,Y 215.533,Z 501.291,A -85,B 0,C 180,E1 -20797.025,E2 -20797.025} C_VEL
LIN {X 0,Y 217.346,Z 493.029,A -85,B 0,C 180,E1 -20799.775,E2 -20799.775} C_VEL
LIN {X 0,Y 219.213,Z 484.521,A -85,B 0,C 180,E1 -20802.029,E2 -20802.029} C_VEL
LIN {X 0,Y 221.331,Z 474.034,A -85,B 0,C 180,E1 -20804.247,E2 -20804.247} C_VEL
LIN {X 0,Y 223.237,Z 463.637,A -85,B 0,C 180,E1 -20805.991,E2 -20805.991} C_VEL
LIN {X 0,Y 224.939,Z 452.227,A -85,B 0,C 180,E1 -20807.502,E2 -20807.502} C_VEL
LIN {X 0,Y 226.32,Z 440.426,A -85,B 0,C 180,E1 -20808.678,E2 -20808.678} C_VEL
LIN {X 0,Y 227.484,Z 426.8,A -85,B 0,C 180,E1 -20809.633,E2 -20809.633} C_VEL
LIN {X 0,Y 228.084,Z 414.563,A -85,B 0,C 180,E1 -20810.165,E2 -20810.165} C_VEL
LIN {X 0,Y 230.309,Z 354.41,A -85,B 0,C 180,E1 -20811.96,E2 -20811.96} C_VEL
LIN {X 0,Y 226.406,Z 344.463,A -85,B 0,C 180,E1 -20812.828,E2 -20812.828} C_VEL
LIN {X 0,Y 219.605,Z 330.497,A -85,B 0,C 180,E1 -20814.303,E2 -20814.303} C_VEL
LIN {X 0,Y 213.977,Z 319.685,A -85,B 0,C 180,E1 -20815.584,E2 -20815.584} C_VEL
LIN {X 0,Y 213.825,Z 318.834,A -85,B 0,C 180,E1 -20815.688,E2 -20815.688} C_VEL
LIN {X 0,Y 213.755,Z 318.856,A -85,B 0,C 180,E1 -20819.551,E2 -20819.551} C_VEL
LIN {X 0,Y 213.759,Z 318.857,A -85,B 0,C 180,E1 -20823.983,E2 -20823.983} C_VEL
LIN {X 0,Y 213.709,Z 318.864,A -85,B 0,C 180,E1 -20828.671,E2 -20828.671} C_VEL
LIN {X 0,Y 213.706,Z 318.864,A -85,B 0,C 180,E1 -20833.655,E2 -20833.655} C_VEL
LIN {X 0,Y 213.706,Z 318.856,A -85,B 0,C 180,E1 -20836.346,E2 -20836.346} C_VEL
LIN {X 0,Y 213.708,Z 318.864,A -85,B 0,C 180,E1 -20841.329,E2 -20841.329} C_VEL
LIN {X 0,Y 213.759,Z 318.842,A -85,B 0,C 180,E1 -20846.017,E2 -20846.017} C_VEL
LIN {X 0,Y 213.754,Z 318.857,A -85,B 0,C 180,E1 -20850.449,E2 -20850.449} C_VEL
LIN {X 0,Y 213.772,Z 318.833,A -85,B 0,C 180,E1 -20854.697,E2 -20854.697} C_VEL
LIN {X 0,Y 213.803,Z 318.851,A -85,B 0,C 180,E1 -20858.802,E2 -20858.802} C_VEL
LIN {X 0,Y 213.927,Z 318.826,A -85,B 0,C 180,E1 -20862.802,E2 -20862.802} C_VEL
LIN {X 0,Y 213.942,Z 318.824,A -85,B 0,C 180,E1 -20866.705,E2 -20866.705} C_VEL
LIN {X 0,Y 214.141,Z 318.809,A -85,B 0,C 180,E1 -20870.555,E2 -20870.555} C_VEL
LIN {X 0,Y 214.079,Z 318.796,A -85,B 0,C 180,E1 -20874.347,E2 -20874.347} C_VEL
LIN {X 0,Y 214.409,Z 318.767,A -85,B 0,C 180,E1 -20878.121,E2 -20878.121} C_VEL
LIN {X 0,Y 214.517,Z 318.762,A -85,B 0,C 180,E1 -20880,E2 -20880} C_VEL
LIN {X 0,Y 214.409,Z 318.776,A -85,B 0,C 180,E1 -20881.878,E2 -20881.878} C_VEL
LIN {X 0,Y 214.184,Z 318.789,A -85,B 0,C 180,E1 -20887.541,E2 -20887.541} C_VEL
LIN {X 0,Y 213.997,Z 318.827,A -85,B 0,C 180,E1 -20891.364,E2 -20891.364} C_VEL
LIN {X 0,Y 213.903,Z 318.84,A -85,B 0,C 180,E1 -20895.239,E2 -20895.239} C_VEL
LIN {X 0,Y 213.8,Z 318.853,A -85,B 0,C 180,E1 -20899.191,E2 -20899.191} C_VEL
LIN {X 0,Y 213.798,Z 318.852,A -85,B 0,C 180,E1 -20903.232,E2 -20903.232} C_VEL
LIN {X 0,Y 213.788,Z 318.854,A -85,B 0,C 180,E1 -20907.426,E2 -20907.426} C_VEL
LIN {X 0,Y 213.762,Z 318.858,A -85,B 0,C 180,E1 -20911.738,E2 -20911.738} C_VEL
LIN {X 0,Y 213.744,Z 318.861,A -85,B 0,C 180,E1 -20916.288,E2 -20916.288} C_VEL
LIN {X 0,Y 213.7,Z 318.868,A -85,B 0,C 180,E1 -20921.128,E2 -20921.128} C_VEL
LIN {X 0,Y 213.704,Z 318.866,A -85,B 0,C 180,E1 -20923.679,E2 -20923.679} C_VEL
LIN {X 0,Y 213.651,Z 318.86,A -85,B 0,C 180,E1 -20927.84,E2 -20927.84} C_VEL
LIN {X 0,Y 213.089,Z 319.321,A -85,B 0,C 180,E1 -20928.889,E2 -20928.889} C_VEL
LIN {X 0,Y 211.291,Z 320.98,A -85,B 0,C 180,E1 -20930.187,E2 -20930.187} C_VEL
LIN {X 0,Y 208.687,Z 324.781,A -85,B 0,C 180,E1 -20932.053,E2 -20932.053} C_VEL
LIN {X 0,Y 208.507,Z 326.907,A -85,B 0,C 180,E1 -20933.01,E2 -20933.01} C_VEL
LIN {X 0,Y 209.25,Z 330.072,A -85,B 0,C 180,E1 -20934.411,E2 -20934.411} C_VEL
LIN {X 0,Y 216.697,Z 348.106,A -85,B 0,C 180,E1 -20936.283,E2 -20936.283} C_VEL
LIN {X 0,Y 219.427,Z 355.66,A -85,B 0,C 180,E1 -20936.964,E2 -20936.964} C_VEL
LIN {X 0,Y 222.357,Z 382.443,A -85,B 0,C 180,E1 -20938.343,E2 -20938.343} C_VEL
LIN {X 0,Y 222.918,Z 388.875,A -85,B 0,C 180,E1 -20938.648,E2 -20938.648} C_VEL
LIN {X 0,Y 221.052,Z 439.842,A -85,B 0,C 180,E1 -20940.278,E2 -20940.278} C_VEL
LIN {X 0,Y 219.784,Z 453.739,A -85,B 0,C 180,E1 -20941.075,E2 -20941.075} C_VEL
LIN {X 0,Y 218.141,Z 466.179,A -85,B 0,C 180,E1 -20942.149,E2 -20942.149} C_VEL
LIN {X 0,Y 216.07,Z 478.902,A -85,B 0,C 180,E1 -20943.692,E2 -20943.692} C_VEL
LIN {X 0,Y 213.834,Z 490.212,A -85,B 0,C 180,E1 -20945.483,E2 -20945.483} C_VEL
LIN {X 0,Y 211.653,Z 500.384,A -85,B 0,C 180,E1 -20947.55,E2 -20947.55} C_VEL
LIN {X 0,Y 209.632,Z 509.62,A -85,B 0,C 180,E1 -20949.914,E2 -20949.914} C_VEL
LIN {X 0,Y 208.055,Z 517.166,A -85,B 0,C 180,E1 -20952.3,E2 -20952.3} C_VEL
LIN {X 0,Y 206.487,Z 524.603,A -85,B 0,C 180,E1 -20955.209,E2 -20955.209} C_VEL
LIN {X 0,Y 205.373,Z 530.56,A -85,B 0,C 180,E1 -20958.15,E2 -20958.15} C_VEL
LIN {X 0,Y 204.781,Z 535.253,A -85,B 0,C 180,E1 -20961.115,E2 -20961.115} C_VEL
LIN {X 0,Y 204.497,Z 538.808,A -85,B 0,C 180,E1 -20964.081,E2 -20964.081} C_VEL
LIN {X 0,Y 204.476,Z 540.603,A -85,B 0,C 180,E1 -20966.057,E2 -20966.057} C_VEL
LIN {X 0,Y 204.58,Z 541.955,A -85,B 0,C 180,E1 -20968.03,E2 -20968.03} C_VEL
LIN {X 0,Y 204.672,Z 542.898,A -85,B 0,C 180,E1 -20969.999,E2 -20969.999} C_VEL
LIN {X 0,Y 204.533,Z 543.432,A -85,B 0,C 180,E1 -20971.968,E2 -20971.968} C_VEL
LIN {X 0,Y 204.438,Z 543.483,A -85,B 0,C 180,E1 -20974.486,E2 -20974.486} C_VEL
LIN {X 0,Y 204.592,Z 542.555,A -85,B 0,C 180,E1 -20977.896,E2 -20977.896} C_VEL
LIN {X 0,Y 204.962,Z 541.491,A -85,B 0,C 180,E1 -20979.871,E2 -20979.871} C_VEL
LIN {X 0,Y 205.518,Z 540.011,A -85,B 0,C 180,E1 -20981.839,E2 -20981.839} C_VEL
LIN {X 0,Y 206.746,Z 536.992,A -85,B 0,C 180,E1 -20984.769,E2 -20984.769} C_VEL
LIN {X 0,Y 208.655,Z 532.948,A -85,B 0,C 180,E1 -20987.645,E2 -20987.645} C_VEL
LIN {X 0,Y 211.422,Z 526.766,A -85,B 0,C 180,E1 -20990.936,E2 -20990.936} C_VEL
LIN {X 0,Y 214.197,Z 520.061,A -85,B 0,C 180,E1 -20993.698,E2 -20993.698} C_VEL
LIN {X 0,Y 217.648,Z 511.774,A -85,B 0,C 180,E1 -20996.358,E2 -20996.358} C_VEL
LIN {X 0,Y 220.974,Z 503.292,A -85,B 0,C 180,E1 -20998.493,E2 -20998.493} C_VEL
LIN {X 0,Y 224.58,Z 492.841,A -85,B 0,C 180,E1 -21000.564,E2 -21000.564} C_VEL
LIN {X 0,Y 227.779,Z 482.519,A -85,B 0,C 180,E1 -21002.156,E2 -21002.156} C_VEL
LIN {X 0,Y 230.672,Z 471.229,A -85,B 0,C 180,E1 -21003.518,E2 -21003.518} C_VEL
LIN {X 0,Y 233.114,Z 459.705,A -85,B 0,C 180,E1 -21004.551,E2 -21004.551} C_VEL
LIN {X 0,Y 235.187,Z 446.184,A -85,B 0,C 180,E1 -21005.4,E2 -21005.4} C_VEL
LIN {X 0,Y 236.338,Z 433.409,A -85,B 0,C 180,E1 -21005.914,E2 -21005.914} C_VEL
LIN {X 0,Y 238.318,Z 393.9,A -85,B 0,C 180,E1 -21007.054,E2 -21007.054} C_VEL
LIN {X 0,Y 236.237,Z 378.681,A -85,B 0,C 180,E1 -21008.094,E2 -21008.094} C_VEL
LIN {X 0,Y 230.217,Z 364.833,A -85,B 0,C 180,E1 -21010.024,E2 -21010.024} C_VEL
LIN {X 0,Y 224.191,Z 352.81,A -85,B 0,C 180,E1 -21012.051,E2 -21012.051} C_VEL
LIN {X 0,Y 218.761,Z 343.212,A -85,B 0,C 180,E1 -21013.984,E2 -21013.984} C_VEL
LIN {X 0,Y 215.475,Z 337.83,A -85,B 0,C 180,E1 -21015.22,E2 -21015.22} C_VEL
LIN {X 0,Y 212.459,Z 333.031,A -85,B 0,C 180,E1 -21016.41,E2 -21016.41} C_VEL
LIN {X 0,Y 209.557,Z 328.619,A -85,B 0,C 180,E1 -21017.608,E2 -21017.608} C_VEL
LIN {X 0,Y 209.137,Z 327.591,A -85,B 0,C 180,E1 -21017.919,E2 -21017.919} C_VEL
LIN {X 0,Y 207.667,Z 322.827,A -85,B 0,C 180,E1 -21021.11,E2 -21021.11} C_VEL
LIN {X 0,Y 206.691,Z 319.738,A -85,B 0,C 180,E1 -21023.485,E2 -21023.485} C_VEL
LIN {X 0,Y 206.714,Z 319.725,A -85,B 0,C 180,E1 -21028.206,E2 -21028.206} C_VEL
LIN {X 0,Y 206.763,Z 319.718,A -85,B 0,C 180,E1 -21032.096,E2 -21032.096} C_VEL
LIN {X 0,Y 206.787,Z 319.717,A -85,B 0,C 180,E1 -21036.58,E2 -21036.58} C_VEL
LIN {X 0,Y 206.87,Z 319.714,A -85,B 0,C 180,E1 -21042.197,E2 -21042.197} C_VEL
LIN {X 0,Y 206.912,Z 319.71,A -85,B 0,C 180,E1 -21046.246,E2 -21046.246} C_VEL
LIN {X 0,Y 207.13,Z 319.685,A -85,B 0,C 180,E1 -21050.233,E2 -21050.233} C_VEL
LIN {X 0,Y 207.072,Z 319.691,A -85,B 0,C 180,E1 -21054.156,E2 -21054.156} C_VEL
LIN {X 0,Y 207.38,Z 319.651,A -85,B 0,C 180,E1 -21058.058,E2 -21058.058} C_VEL
LIN {X 0,Y 207.512,Z 319.627,A -85,B 0,C 180,E1 -21060,E2 -21060} C_VEL
LIN {X 0,Y 207.38,Z 319.648,A -85,B 0,C 180,E1 -21061.943,E2 -21061.943} C_VEL
LIN {X 0,Y 207.186,Z 319.674,A -85,B 0,C 180,E1 -21067.799,E2 -21067.799} C_VEL
LIN {X 0,Y 206.981,Z 319.701,A -85,B 0,C 180,E1 -21071.756,E2 -21071.756} C_VEL
LIN {X 0,Y 206.865,Z 319.716,A -85,B 0,C 180,E1 -21075.771,E2 -21075.771} C_VEL
LIN {X 0,Y 206.797,Z 319.725,A -85,B 0,C 180,E1 -21079.868,E2 -21079.868} C_VEL
LIN {X 0,Y 206.761,Z 319.727,A -85,B 0,C 180,E1 -21084.073,E2 -21084.073} C_VEL
LIN {X 0,Y 206.735,Z 319.725,A -85,B 0,C 180,E1 -21088.421,E2 -21088.421} C_VEL
LIN {X 0,Y 206.705,Z 319.829,A -85,B 0,C 180,E1 -21092.581,E2 -21092.581} C_VEL
LIN {X 0,Y 207.544,Z 322.308,A -85,B 0,C 180,E1 -21093.024,E2 -21093.024} C_VEL
LIN {X 0,Y 209.358,Z 324.44,A -85,B 0,C 180,E1 -21093.78,E2 -21093.78} C_VEL
LIN {X 0,Y 210.375,Z 325.243,A -85,B 0,C 180,E1 -21094.171,E2 -21094.171} C_VEL
LIN {X 0,Y 212.344,Z 328.441,A -85,B 0,C 180,E1 -21094.995,E2 -21094.995} C_VEL
LIN {X 0,Y 214.063,Z 330.354,A -85,B 0,C 180,E1 -21095.646,E2 -21095.646} C_VEL
LIN {X 0,Y 216.582,Z 333.925,A -85,B 0,C 180,E1 -21096.603,E2 -21096.603} C_VEL
LIN {X 0,Y 223.356,Z 343.795,A -85,B 0,C 180,E1 -21099,E2 -21099} C_VEL
LIN {X 0,Y 231.221,Z 356.386,A -85,B 0,C 180,E1 -21101.538,E2 -21101.538} C_VEL
LIN {X 0,Y 236.725,Z 366.65,A -85,B 0,C 180,E1 -21103.212,E2 -21103.212} C_VEL
LIN {X 0,Y 239.443,Z 372.498,A -85,B 0,C 180,E1 -21104.024,E2 -21104.024} C_VEL
LIN {X 0,Y 236.737,Z 421.247,A -85,B 0,C 180,E1 -21105.417,E2 -21105.417} C_VEL
LIN {X 0,Y 235.394,Z 434.852,A -85,B 0,C 180,E1 -21106.142,E2 -21106.142} C_VEL
LIN {X 0,Y 233.502,Z 446.974,A -85,B 0,C 180,E1 -21107.082,E2 -21107.082} C_VEL
LIN {X 0,Y 230.918,Z 458.533,A -85,B 0,C 180,E1 -21108.26,E2 -21108.26} C_VEL
LIN {X 0,Y 227.874,Z 470.243,A -85,B 0,C 180,E1 -21109.896,E2 -21109.896} C_VEL
LIN {X 0,Y 224.774,Z 480.977,A -85,B 0,C 180,E1 -21111.866,E2 -21111.866} C_VEL
LIN {X 0,Y 221.382,Z 490.429,A -85,B 0,C 180,E1 -21114.036,E2 -21114.036} C_VEL
LIN {X 0,Y 217.729,Z 499.518,A -85,B 0,C 180,E1 -21116.721,E2 -21116.721} C_VEL
LIN {X 0,Y 214.583,Z 506.797,A -85,B 0,C 180,E1 -21119.494,E2 -21119.494} C_VEL
LIN {X 0,Y 211.77,Z 512.554,A -85,B 0,C 180,E1 -21122.316,E2 -21122.316} C_VEL
LIN {X 0,Y 209.876,Z 516.351,A -85,B 0,C 180,E1 -21124.709,E2 -21124.709} C_VEL
LIN {X 0,Y 207.673,Z 520.425,A -85,B 0,C 180,E1 -21128.146,E2 -21128.146} C_VEL
LIN {X 0,Y 206.711,Z 522.086,A -85,B 0,C 180,E1 -21130.125,E2 -21130.125} C_VEL
LIN {X 0,Y 205.64,Z 523.8,A -85,B 0,C 180,E1 -21133.127,E2 -21133.127} C_VEL
LIN {X 0,Y 204.877,Z 524.581,A -85,B 0,C 180,E1 -21136.107,E2 -21136.107} C_VEL
LIN {X 0,Y 204.434,Z 524.207,A -85,B 0,C 180,E1 -21140.104,E2 -21140.104} C_VEL
LIN {X 0,Y 204.441,Z 523.433,A -85,B 0,C 180,E1 -21142.098,E2 -21142.098} C_VEL
LIN {X 0,Y 204.711,Z 521.803,A -85,B 0,C 180,E1 -21144.638,E2 -21144.638} C_VEL
LIN {X 0,Y 205.049,Z 518.586,A -85,B 0,C 180,E1 -21148.037,E2 -21148.037} C_VEL
LIN {X 0,Y 205.786,Z 514.668,A -85,B 0,C 180,E1 -21150.98,E2 -21150.98} C_VEL
LIN {X 0,Y 206.826,Z 509.629,A -85,B 0,C 180,E1 -21153.898,E2 -21153.898} C_VEL
LIN {X 0,Y 208.228,Z 503.295,A -85,B 0,C 180,E1 -21156.785,E2 -21156.785} C_VEL
LIN {X 0,Y 210.026,Z 495.381,A -85,B 0,C 180,E1 -21159.633,E2 -21159.633} C_VEL
LIN {X 0,Y 212.305,Z 485.539,A -85,B 0,C 180,E1 -21162.427,E2 -21162.427} C_VEL
LIN {X 0,Y 214.508,Z 475.216,A -85,B 0,C 180,E1 -21164.711,E2 -21164.711} C_VEL
LIN {X 0,Y 216.728,Z 463.585,A -85,B 0,C 180,E1 -21166.727,E2 -21166.727} C_VEL
LIN {X 0,Y 218.494,Z 452.039,A -85,B 0,C 180,E1 -21168.278,E2 -21168.278} C_VEL
LIN {X 0,Y 219.952,Z 440.061,A -85,B 0,C 180,E1 -21169.483,E2 -21169.483} C_VEL
LIN {X 0,Y 221.073,Z 427.072,A -85,B 0,C 180,E1 -21170.409,E2 -21170.409} C_VEL
LIN {X 0,Y 221.719,Z 414.776,A -85,B 0,C 180,E1 -21170.952,E2 -21170.952} C_VEL
LIN {X 0,Y 224.017,Z 356.047,A -85,B 0,C 180,E1 -21172.742,E2 -21172.742} C_VEL
LIN {X 0,Y 220.019,Z 346.202,A -85,B 0,C 180,E1 -21173.663,E2 -21173.663} C_VEL
LIN {X 0,Y 212.498,Z 331.044,A -85,B 0,C 180,E1 -21175.383,E2 -21175.383} C_VEL
LIN {X 0,Y 207.766,Z 322.481,A -85,B 0,C 180,E1 -21176.507,E2 -21176.507} C_VEL
LIN {X 0,Y 206.778,Z 319.72,A -85,B 0,C 180,E1 -21176.82,E2 -21176.82} C_VEL
LIN {X 0,Y 206.714,Z 319.735,A -85,B 0,C 180,E1 -21181.79,E2 -21181.79} C_VEL
LIN {X 0,Y 206.704,Z 319.738,A -85,B 0,C 180,E1 -21185.312,E2 -21185.312} C_VEL
LIN {X 0,Y 206.652,Z 319.735,A -85,B 0,C 180,E1 -21190.255,E2 -21190.255} C_VEL
LIN {X 0,Y 206.634,Z 319.743,A -85,B 0,C 180,E1 -21194.417,E2 -21194.417} C_VEL
LIN {X 0,Y 206.635,Z 319.732,A -85,B 0,C 180,E1 -21198.442,E2 -21198.442} C_VEL
LIN {X 0,Y 206.672,Z 319.737,A -85,B 0,C 180,E1 -21202.258,E2 -21202.258} C_VEL
LIN {X 0,Y 206.699,Z 319.726,A -85,B 0,C 180,E1 -21207.042,E2 -21207.042} C_VEL
LIN {X 0,Y 206.713,Z 319.728,A -85,B 0,C 180,E1 -21212.128,E2 -21212.128} C_VEL
LIN {X 0,Y 206.746,Z 319.722,A -85,B 0,C 180,E1 -21216.613,E2 -21216.613} C_VEL
LIN {X 0,Y 206.873,Z 319.706,A -85,B 0,C 180,E1 -21222.196,E2 -21222.196} C_VEL
LIN {X 0,Y 206.884,Z 319.696,A -85,B 0,C 180,E1 -21226.243,E2 -21226.243} C_VEL
LIN {X 0,Y 207.085,Z 319.689,A -85,B 0,C 180,E1 -21230.23,E2 -21230.23} C_VEL
LIN {X 0,Y 207.043,Z 319.673,A -85,B 0,C 180,E1 -21234.155,E2 -21234.155} C_VEL
LIN {X 0,Y 207.348,Z 319.646,A -85,B 0,C 180,E1 -21238.057,E2 -21238.057} C_VEL
LIN {X 0,Y 207.484,Z 319.638,A -85,B 0,C 180,E1 -21240,E2 -21240} C_VEL
LIN {X 0,Y 207.349,Z 319.656,A -85,B 0,C 180,E1 -21241.942,E2 -21241.942} C_VEL
LIN {X 0,Y 207.129,Z 319.667,A -85,B 0,C 180,E1 -21247.8,E2 -21247.8} C_VEL
LIN {X 0,Y 206.919,Z 319.709,A -85,B 0,C 180,E1 -21251.758,E2 -21251.758} C_VEL
LIN {X 0,Y 206.83,Z 319.72,A -85,B 0,C 180,E1 -21255.773,E2 -21255.773} C_VEL
LIN {X 0,Y 206.721,Z 319.734,A -85,B 0,C 180,E1 -21259.875,E2 -21259.875} C_VEL
LIN {X 0,Y 206.738,Z 319.732,A -85,B 0,C 180,E1 -21264.075,E2 -21264.075} C_VEL
LIN {X 0,Y 206.691,Z 319.739,A -85,B 0,C 180,E1 -21268.426,E2 -21268.426} C_VEL
LIN {X 0,Y 206.697,Z 319.742,A -85,B 0,C 180,E1 -21272.958,E2 -21272.958} C_VEL
LIN {X 0,Y 206.671,Z 319.743,A -85,B 0,C 180,E1 -21277.741,E2 -21277.741} C_VEL
LIN {X 0,Y 206.634,Z 319.747,A -85,B 0,C 180,E1 -21281.558,E2 -21281.558} C_VEL
LIN {X 0,Y 206.632,Z 319.745,A -85,B 0,C 180,E1 -21285.582,E2 -21285.582} C_VEL
LIN {X 0,Y 206.704,Z 319.779,A -85,B 0,C 180,E1 -21289.625,E2 -21289.625} C_VEL
LIN {X 0,Y 208.507,Z 326.907,A -85,B 0,C 180,E1 -21293.01,E2 -21293.01} C_VEL
LIN {X 0,Y 209.035,Z 329.393,A -85,B 0,C 180,E1 -21293.789,E2 -21293.789} C_VEL
LIN {X 0,Y 209.772,Z 333.475,A -85,B 0,C 180,E1 -21294.466,E2 -21294.466} C_VEL
LIN {X 0,Y 210.627,Z 340.027,A -85,B 0,C 180,E1 -21295.028,E2 -21295.028} C_VEL
LIN {X 0,Y 211.855,Z 352.338,A -85,B 0,C 180,E1 -21295.7,E2 -21295.7} C_VEL
LIN {X 0,Y 212.834,Z 356.237,A -85,B 0,C 180,E1 -21296.003,E2 -21296.003} C_VEL
LIN {X 0,Y 213.514,Z 359.029,A -85,B 0,C 180,E1 -21296.214,E2 -21296.214} C_VEL
LIN {X 0,Y 216.269,Z 385.286,A -85,B 0,C 180,E1 -21297.606,E2 -21297.606} C_VEL
LIN {X 0,Y 216.542,Z 391.481,A -85,B 0,C 180,E1 -21297.873,E2 -21297.873} C_VEL
LIN {X 0,Y 214.706,Z 439.341,A -85,B 0,C 180,E1 -21299.442,E2 -21299.442} C_VEL
LIN {X 0,Y 213.406,Z 453.301,A -85,B 0,C 180,E1 -21300.26,E2 -21300.26} C_VEL
LIN {X 0,Y 211.7,Z 465.777,A -85,B 0,C 180,E1 -21301.359,E2 -21301.359} C_VEL
LIN {X 0,Y 209.653,Z 477.712,A -85,B 0,C 180,E1 -21302.822,E2 -21302.822} C_VEL
LIN {X 0,Y 207.281,Z 489.175,A -85,B 0,C 180,E1 -21304.654,E2 -21304.654} C_VEL
LIN {X 0,Y 205.009,Z 499.517,A -85,B 0,C 180,E1 -21306.78,E2 -21306.78} C_VEL
LIN {X 0,Y 202.908,Z 508.975,A -85,B 0,C 180,E1 -21309.257,E2 -21309.257} C_VEL
LIN {X 0,Y 201.283,Z 516.476,A -85,B 0,C 180,E1 -21311.684,E2 -21311.684} C_VEL
LIN {X 0,Y 199.607,Z 523.976,A -85,B 0,C 180,E1 -21314.687,E2 -21314.687} C_VEL
LIN {X 0,Y 198.376,Z 529.986,A -85,B 0,C 180,E1 -21317.726,E2 -21317.726} C_VEL
LIN {X 0,Y 197.723,Z 534.73,A -85,B 0,C 180,E1 -21320.795,E2 -21320.795} C_VEL
LIN {X 0,Y 197.41,Z 538.335,A -85,B 0,C 180,E1 -21323.868,E2 -21323.868} C_VEL
LIN {X 0,Y 197.413,Z 540.178,A -85,B 0,C 180,E1 -21325.916,E2 -21325.916} C_VEL
LIN {X 0,Y 197.492,Z 541.55,A -85,B 0,C 180,E1 -21327.959,E2 -21327.959} C_VEL
LIN {X 0,Y 197.605,Z 542.517,A -85,B 0,C 180,E1 -21329.999,E2 -21329.999} C_VEL
LIN {X 0,Y 197.446,Z 543.07,A -85,B 0,C 180,E1 -21332.039,E2 -21332.039} C_VEL
LIN {X 0,Y 197.338,Z 543.196,A -85,B 0,C 180,E1 -21334.297,E2 -21334.297} C_VEL
LIN {X 0,Y 197.527,Z 542.276,A -85,B 0,C 180,E1 -21338.181,E2 -21338.181} C_VEL
LIN {X 0,Y 198.542,Z 539.793,A -85,B 0,C 180,E1 -21342.261,E2 -21342.261} C_VEL
LIN {X 0,Y 199.858,Z 536.81,A -85,B 0,C 180,E1 -21345.291,E2 -21345.291} C_VEL
LIN {X 0,Y 201.859,Z 532.813,A -85,B 0,C 180,E1 -21348.26,E2 -21348.26} C_VEL
LIN {X 0,Y 204.784,Z 526.707,A -85,B 0,C 180,E1 -21351.648,E2 -21351.648} C_VEL
LIN {X 0,Y 207.691,Z 520.063,A -85,B 0,C 180,E1 -21354.488,E2 -21354.488} C_VEL
LIN {X 0,Y 211.318,Z 511.844,A -85,B 0,C 180,E1 -21357.211,E2 -21357.211} C_VEL
LIN {X 0,Y 214.771,Z 503.459,A -85,B 0,C 180,E1 -21359.395,E2 -21359.395} C_VEL
LIN {X 0,Y 218.517,Z 493.144,A -85,B 0,C 180,E1 -21361.508,E2 -21361.508} C_VEL
LIN {X 0,Y 221.826,Z 482.958,A -85,B 0,C 180,E1 -21363.127,E2 -21363.127} C_VEL
LIN {X 0,Y 224.812,Z 471.852,A -85,B 0,C 180,E1 -21364.513,E2 -21364.513} C_VEL
LIN {X 0,Y 227.563,Z 459.48,A -85,B 0,C 180,E1 -21365.656,E2 -21365.656} C_VEL
LIN {X 0,Y 229.703,Z 445.996,A -85,B 0,C 180,E1 -21366.515,E2 -21366.515} C_VEL
LIN {X 0,Y 230.864,Z 433.797,A -85,B 0,C 180,E1 -21367.02,E2 -21367.02} C_VEL
LIN {X 0,Y 232.926,Z 395.059,A -85,B 0,C 180,E1 -21368.153,E2 -21368.153} C_VEL
LIN {X 0,Y 231.108,Z 381.498,A -85,B 0,C 180,E1 -21369.116,E2 -21369.116} C_VEL
LIN {X 0,Y 225.356,Z 368.156,A -85,B 0,C 180,E1 -21371.068,E2 -21371.068} C_VEL
LIN {X 0,Y 219.883,Z 357.099,A -85,B 0,C 180,E1 -21373.012,E2 -21373.012} C_VEL
LIN {X 0,Y 214.853,Z 348.09,A -85,B 0,C 180,E1 -21374.898,E2 -21374.898} C_VEL
LIN {X 0,Y 210.983,Z 341.648,A -85,B 0,C 180,E1 -21376.44,E2 -21376.44} C_VEL
LIN {X 0,Y 209.054,Z 338.447,A -85,B 0,C 180,E1 -21377.249,E2 -21377.249} C_VEL
LIN {X 0,Y 205.97,Z 333.581,A -85,B 0,C 180,E1 -21378.593,E2 -21378.593} C_VEL
LIN {X 0,Y 202.179,Z 328.164,A -85,B 0,C 180,E1 -21380.329,E2 -21380.329} C_VEL
LIN {X 0,Y 201.688,Z 327.028,A -85,B 0,C 180,E1 -21380.696,E2 -21380.696} C_VEL
LIN {X 0,Y 200.068,Z 322.26,A -85,B 0,C 180,E1 -21384.321,E2 -21384.321} C_VEL
LIN {X 0,Y 199.608,Z 320.611,A -85,B 0,C 180,E1 -21385.713,E2 -21385.713} C_VEL
LIN {X 0,Y 199.69,Z 320.6,A -85,B 0,C 180,E1 -21388.135,E2 -21388.135} C_VEL
LIN {X 0,Y 199.684,Z 320.601,A -85,B 0,C 180,E1 -21392.772,E2 -21392.772} C_VEL
LIN {X 0,Y 199.743,Z 320.6,A -85,B 0,C 180,E1 -21397.23,E2 -21397.23} C_VEL
LIN {X 0,Y 199.794,Z 320.598,A -85,B 0,C 180,E1 -21401.757,E2 -21401.757} C_VEL
LIN {X 0,Y 199.847,Z 320.592,A -85,B 0,C 180,E1 -21405.75,E2 -21405.75} C_VEL
LIN {X 0,Y 200.072,Z 320.564,A -85,B 0,C 180,E1 -21409.885,E2 -21409.885} C_VEL
LIN {X 0,Y 200.035,Z 320.567,A -85,B 0,C 180,E1 -21413.95,E2 -21413.95} C_VEL
LIN {X 0,Y 200.319,Z 320.531,A -85,B 0,C 180,E1 -21417.99,E2 -21417.99} C_VEL
LIN {X 0,Y 200.477,Z 320.503,A -85,B 0,C 180,E1 -21420.001,E2 -21420.001} C_VEL
LIN {X 0,Y 200.029,Z 320.56,A -85,B 0,C 180,E1 -21424.03,E2 -21424.03} C_VEL
LIN {X 0,Y 200.129,Z 320.549,A -85,B 0,C 180,E1 -21428.076,E2 -21428.076} C_VEL
LIN {X 0,Y 199.912,Z 320.578,A -85,B 0,C 180,E1 -21432.178,E2 -21432.178} C_VEL
LIN {X 0,Y 199.804,Z 320.591,A -85,B 0,C 180,E1 -21436.344,E2 -21436.344} C_VEL
LIN {X 0,Y 199.821,Z 320.587,A -85,B 0,C 180,E1 -21438.455,E2 -21438.455} C_VEL
LIN {X 0,Y 199.735,Z 320.605,A -85,B 0,C 180,E1 -21443.818,E2 -21443.818} C_VEL
LIN {X 0,Y 199.706,Z 320.601,A -85,B 0,C 180,E1 -21448.385,E2 -21448.385} C_VEL
LIN {X 0,Y 199.674,Z 320.719,A -85,B 0,C 180,E1 -21449.886,E2 -21449.886} C_VEL
LIN {X 0,Y 200.426,Z 323.054,A -85,B 0,C 180,E1 -21450.343,E2 -21450.343} C_VEL
LIN {X 0,Y 202.35,Z 325.338,A -85,B 0,C 180,E1 -21451.253,E2 -21451.253} C_VEL
LIN {X 0,Y 203.525,Z 326.28,A -85,B 0,C 180,E1 -21451.764,E2 -21451.764} C_VEL
LIN {X 0,Y 205.576,Z 329.587,A -85,B 0,C 180,E1 -21452.721,E2 -21452.721} C_VEL
LIN {X 0,Y 207.361,Z 331.421,A -85,B 0,C 180,E1 -21453.465,E2 -21453.465} C_VEL
LIN {X 0,Y 210.016,Z 335.106,A -85,B 0,C 180,E1 -21454.577,E2 -21454.577} C_VEL
LIN {X 0,Y 216.315,Z 343.991,A -85,B 0,C 180,E1 -21457.019,E2 -21457.019} C_VEL
LIN {X 0,Y 223.655,Z 355.495,A -85,B 0,C 180,E1 -21459.611,E2 -21459.611} C_VEL
LIN {X 0,Y 229.947,Z 366.36,A -85,B 0,C 180,E1 -21461.658,E2 -21461.658} C_VEL
LIN {X 0,Y 233.986,Z 374.817,A -85,B 0,C 180,E1 -21462.94,E2 -21462.94} C_VEL
LIN {X 0,Y 231.275,Z 422.098,A -85,B 0,C 180,E1 -21464.326,E2 -21464.326} C_VEL
LIN {X 0,Y 229.878,Z 435.515,A -85,B 0,C 180,E1 -21465.061,E2 -21465.061} C_VEL
LIN {X 0,Y 227.828,Z 447.95,A -85,B 0,C 180,E1 -21466.048,E2 -21466.048} C_VEL
LIN {X 0,Y 225.145,Z 459.318,A -85,B 0,C 180,E1 -21467.241,E2 -21467.241} C_VEL
LIN {X 0,Y 222.279,Z 469.887,A -85,B 0,C 180,E1 -21468.73,E2 -21468.73} C_VEL
LIN {X 0,Y 219.108,Z 480.526,A -85,B 0,C 180,E1 -21470.693,E2 -21470.693} C_VEL
LIN {X 0,Y 215.546,Z 490.157,A -85,B 0,C 180,E1 -21472.902,E2 -21472.902} C_VEL
LIN {X 0,Y 211.702,Z 499.357,A -85,B 0,C 180,E1 -21475.644,E2 -21475.644} C_VEL
LIN {X 0,Y 208.36,Z 506.725,A -85,B 0,C 180,E1 -21478.48,E2 -21478.48} C_VEL
LIN {X 0,Y 205.387,Z 512.583,A -85,B 0,C 180,E1 -21481.378,E2 -21481.378} C_VEL
LIN {X 0,Y 203.121,Z 516.818,A -85,B 0,C 180,E1 -21484.108,E2 -21484.108} C_VEL
LIN {X 0,Y 200.953,Z 520.594,A -85,B 0,C 180,E1 -21487.376,E2 -21487.376} C_VEL
LIN {X 0,Y 199.912,Z 522.289,A -85,B 0,C 180,E1 -21489.419,E2 -21489.419} C_VEL
LIN {X 0,Y 198.418,Z 524.446,A -85,B 0,C 180,E1 -21493.54,E2 -21493.54} C_VEL
LIN {X 0,Y 197.901,Z 524.9,A -85,B 0,C 180,E1 -21495.607,E2 -21495.607} C_VEL
LIN {X 0,Y 197.342,Z 524.586,A -85,B 0,C 180,E1 -21499.744,E2 -21499.744} C_VEL
LIN {X 0,Y 197.357,Z 523.847,A -85,B 0,C 180,E1 -21501.812,E2 -21501.812} C_VEL
LIN {X 0,Y 197.626,Z 522.073,A -85,B 0,C 180,E1 -21504.718,E2 -21504.718} C_VEL
LIN {X 0,Y 198.115,Z 517.941,A -85,B 0,C 180,E1 -21508.985,E2 -21508.985} C_VEL
LIN {X 0,Y 199,Z 513.725,A -85,B 0,C 180,E1 -21512.025,E2 -21512.025} C_VEL
LIN {X 0,Y 200.373,Z 507.345,A -85,B 0,C 180,E1 -21515.536,E2 -21515.536} C_VEL
LIN {X 0,Y 202.073,Z 500.371,A -85,B 0,C 180,E1 -21518.501,E2 -21518.501} C_VEL
LIN {X 0,Y 204.186,Z 491.645,A -85,B 0,C 180,E1 -21521.416,E2 -21521.416} C_VEL
LIN {X 0,Y 206.509,Z 481.74,A -85,B 0,C 180,E1 -21524.034,E2 -21524.034} C_VEL
LIN {X 0,Y 208.667,Z 471.638,A -85,B 0,C 180,E1 -21526.134,E2 -21526.134} C_VEL
LIN {X 0,Y 210.814,Z 460.422,A -85,B 0,C 180,E1 -21527.962,E2 -21527.962} C_VEL
LIN {X 0,Y 212.572,Z 447.881,A -85,B 0,C 180,E1 -21529.559,E2 -21529.559} C_VEL
LIN {X 0,Y 214.123,Z 434.806,A -85,B 0,C 180,E1 -21530.725,E2 -21530.725} C_VEL
LIN {X 0,Y 215.092,Z 421.41,A -85,B 0,C 180,E1 -21531.534,E2 -21531.534} C_VEL
LIN {X 0,Y 217.704,Z 357.666,A -85,B 0,C 180,E1 -21533.577,E2 -21533.577} C_VEL
LIN {X 0,Y 213.1,Z 346.768,A -85,B 0,C 180,E1 -21534.683,E2 -21534.683} C_VEL
LIN {X 0,Y 204.877,Z 330.575,A -85,B 0,C 180,E1 -21536.683,E2 -21536.683} C_VEL
LIN {X 0,Y 201.174,Z 324.137,A -85,B 0,C 180,E1 -21537.616,E2 -21537.616} C_VEL
LIN {X 0,Y 199.848,Z 321.514,A -85,B 0,C 180,E1 -21537.974,E2 -21537.974} C_VEL
LIN {X 0,Y 199.676,Z 320.607,A -85,B 0,C 180,E1 -21538.089,E2 -21538.089} C_VEL
LIN {X 0,Y 199.67,Z 320.613,A -85,B 0,C 180,E1 -21542.353,E2 -21542.353} C_VEL
LIN {X 0,Y 199.622,Z 320.618,A -85,B 0,C 180,E1 -21546.765,E2 -21546.765} C_VEL
LIN {X 0,Y 199.599,Z 320.618,A -85,B 0,C 180,E1 -21549.332,E2 -21549.332} C_VEL
LIN {X 0,Y 199.571,Z 320.618,A -85,B 0,C 180,E1 -21552.308,E2 -21552.308} C_VEL
LIN {X 0,Y 199.581,Z 320.62,A -85,B 0,C 180,E1 -21555.228,E2 -21555.228} C_VEL
LIN {X 0,Y 199.573,Z 320.609,A -85,B 0,C 180,E1 -21558.002,E2 -21558.002} C_VEL
LIN {X 0,Y 199.601,Z 320.619,A -85,B 0,C 180,E1 -21560.773,E2 -21560.773} C_VEL
LIN {X 0,Y 199.615,Z 320.6,A -85,B 0,C 180,E1 -21565.713,E2 -21565.713} C_VEL
LIN {X 0,Y 199.691,Z 320.607,A -85,B 0,C 180,E1 -21568.134,E2 -21568.134} C_VEL
LIN {X 0,Y 199.643,Z 320.606,A -85,B 0,C 180,E1 -21572.765,E2 -21572.765} C_VEL
LIN {X 0,Y 199.709,Z 320.6,A -85,B 0,C 180,E1 -21577.225,E2 -21577.225} C_VEL
LIN {X 0,Y 199.801,Z 320.59,A -85,B 0,C 180,E1 -21581.759,E2 -21581.759} C_VEL
LIN {X 0,Y 199.824,Z 320.57,A -85,B 0,C 180,E1 -21585.747,E2 -21585.747} C_VEL
LIN {X 0,Y 200.028,Z 320.568,A -85,B 0,C 180,E1 -21589.881,E2 -21589.881} C_VEL
LIN {X 0,Y 200.007,Z 320.55,A -85,B 0,C 180,E1 -21593.948,E2 -21593.948} C_VEL
LIN {X 0,Y 200.29,Z 320.524,A -85,B 0,C 180,E1 -21597.989,E2 -21597.989} C_VEL
LIN {X 0,Y 200.452,Z 320.514,A -85,B 0,C 180,E1 -21599.999,E2 -21599.999} C_VEL
LIN {X 0,Y 199.991,Z 320.559,A -85,B 0,C 180,E1 -21604.03,E2 -21604.03} C_VEL
LIN {X 0,Y 200.078,Z 320.546,A -85,B 0,C 180,E1 -21608.077,E2 -21608.077} C_VEL
LIN {X 0,Y 199.869,Z 320.589,A -85,B 0,C 180,E1 -21612.179,E2 -21612.179} C_VEL
LIN {X 0,Y 199.767,Z 320.602,A -85,B 0,C 180,E1 -21616.346,E2 -21616.346} C_VEL
LIN {X 0,Y 199.653,Z 320.617,A -85,B 0,C 180,E1 -21620.61,E2 -21620.61} C_VEL
LIN {X 0,Y 199.652,Z 320.619,A -85,B 0,C 180,E1 -21624.987,E2 -21624.987} C_VEL
LIN {X 0,Y 199.611,Z 320.622,A -85,B 0,C 180,E1 -21629.532,E2 -21629.532} C_VEL
LIN {X 0,Y 199.668,Z 320.615,A -85,B 0,C 180,E1 -21632.351,E2 -21632.351} C_VEL
LIN {X 0,Y 199.62,Z 320.623,A -85,B 0,C 180,E1 -21636.763,E2 -21636.763} C_VEL
LIN {X 0,Y 199.597,Z 320.625,A -85,B 0,C 180,E1 -21639.33,E2 -21639.33} C_VEL
LIN {X 0,Y 199.568,Z 320.626,A -85,B 0,C 180,E1 -21642.306,E2 -21642.306} C_VEL
LIN {X 0,Y 199.578,Z 320.626,A -85,B 0,C 180,E1 -21645.226,E2 -21645.226} C_VEL
LIN {X 0,Y 199.626,Z 320.686,A -85,B 0,C 180,E1 -21648.72,E2 -21648.72} C_VEL
LIN {X 0,Y 201.88,Z 329.543,A -85,B 0,C 180,E1 -21653.093,E2 -21653.093} C_VEL
LIN {X 0,Y 208.982,Z 345.995,A -85,B 0,C 180,E1 -21654.994,E2 -21654.994} C_VEL
LIN {X 0,Y 212.834,Z 356.237,A -85,B 0,C 180,E1 -21656.003,E2 -21656.003} C_VEL
LIN {X 0,Y 213.581,Z 359.928,A -85,B 0,C 180,E1 -21656.258,E2 -21656.258} C_VEL
LIN {X 0,Y 213.591,Z 363.795,A -85,B 0,C 180,E1 -21656.407,E2 -21656.407} C_VEL
LIN {X 0,Y 212.287,Z 371.64,A -85,B 0,C 180,E1 -21656.508,E2 -21656.508} C_VEL
LIN {X 0,Y 210.258,Z 381.629,A -85,B 0,C 180,E1 -21656.583,E2 -21656.583} C_VEL
LIN {X 0,Y 210.155,Z 387.618,A -85,B 0,C 180,E1 -21656.798,E2 -21656.798} C_VEL
LIN {X 0,Y 210.218,Z 394.761,A -85,B 0,C 180,E1 -21657.081,E2 -21657.081} C_VEL
LIN {X 0,Y 208.396,Z 438.857,A -85,B 0,C 180,E1 -21658.557,E2 -21658.557} C_VEL
LIN {X 0,Y 207.156,Z 452.125,A -85,B 0,C 180,E1 -21659.343,E2 -21659.343} C_VEL
LIN {X 0,Y 205.442,Z 464.234,A -85,B 0,C 180,E1 -21660.402,E2 -21660.402} C_VEL
LIN {X 0,Y 203.34,Z 476.519,A -85,B 0,C 180,E1 -21661.905,E2 -21661.905} C_VEL
LIN {X 0,Y 200.879,Z 488.142,A -85,B 0,C 180,E1 -21663.786,E2 -21663.786} C_VEL
LIN {X 0,Y 198.516,Z 498.624,A -85,B 0,C 180,E1 -21665.974,E2 -21665.974} C_VEL
LIN {X 0,Y 196.063,Z 508.941,A -85,B 0,C 180,E1 -21668.746,E2 -21668.746} C_VEL
LIN {X 0,Y 194.142,Z 517.143,A -85,B 0,C 180,E1 -21671.532,E2 -21671.532} C_VEL
LIN {X 0,Y 192.451,Z 524.47,A -85,B 0,C 180,E1 -21674.646,E2 -21674.646} C_VEL
LIN {X 0,Y 191.399,Z 529.408,A -85,B 0,C 180,E1 -21677.271,E2 -21677.271} C_VEL
LIN {X 0,Y 190.686,Z 534.207,A -85,B 0,C 180,E1 -21680.452,E2 -21680.452} C_VEL
LIN {X 0,Y 190.348,Z 537.862,A -85,B 0,C 180,E1 -21683.639,E2 -21683.639} C_VEL
LIN {X 0,Y 190.316,Z 539.742,A -85,B 0,C 180,E1 -21685.763,E2 -21685.763} C_VEL
LIN {X 0,Y 190.408,Z 541.145,A -85,B 0,C 180,E1 -21687.883,E2 -21687.883} C_VEL
LIN {X 0,Y 190.516,Z 542.133,A -85,B 0,C 180,E1 -21689.999,E2 -21689.999} C_VEL
LIN {X 0,Y 190.361,Z 542.707,A -85,B 0,C 180,E1 -21692.114,E2 -21692.114} C_VEL
LIN {X 0,Y 190.244,Z 542.887,A -85,B 0,C 180,E1 -21694.236,E2 -21694.236} C_VEL
LIN {X 0,Y 190.484,Z 541.998,A -85,B 0,C 180,E1 -21698.485,E2 -21698.485} C_VEL
LIN {X 0,Y 191.585,Z 539.567,A -85,B 0,C 180,E1 -21702.714,E2 -21702.714} C_VEL
LIN {X 0,Y 192.992,Z 536.623,A -85,B 0,C 180,E1 -21705.849,E2 -21705.849} C_VEL
LIN {X 0,Y 195.088,Z 532.673,A -85,B 0,C 180,E1 -21708.917,E2 -21708.917} C_VEL
LIN {X 0,Y 197.709,Z 527.614,A -85,B 0,C 180,E1 -21711.914,E2 -21711.914} C_VEL
LIN {X 0,Y 200.691,Z 521.288,A -85,B 0,C 180,E1 -21714.848,E2 -21714.848} C_VEL
LIN {X 0,Y 204.348,Z 513.402,A -85,B 0,C 180,E1 -21717.663,E2 -21717.663} C_VEL
LIN {X 0,Y 208.619,Z 503.61,A -85,B 0,C 180,E1 -21720.351,E2 -21720.351} C_VEL
LIN {X 0,Y 212.521,Z 493.447,A -85,B 0,C 180,E1 -21722.504,E2 -21722.504} C_VEL
LIN {X 0,Y 215.936,Z 483.397,A -85,B 0,C 180,E1 -21724.153,E2 -21724.153} C_VEL
LIN {X 0,Y 219.027,Z 472.475,A -85,B 0,C 180,E1 -21725.56,E2 -21725.56} C_VEL
LIN {X 0,Y 221.869,Z 460.405,A -85,B 0,C 180,E1 -21726.717,E2 -21726.717} C_VEL
LIN {X 0,Y 224.068,Z 447.943,A -85,B 0,C 180,E1 -21727.565,E2 -21727.565} C_VEL
LIN {X 0,Y 225.467,Z 434.489,A -85,B 0,C 180,E1 -21728.167,E2 -21728.167} C_VEL
LIN {X 0,Y 227.64,Z 396.066,A -85,B 0,C 180,E1 -21729.308,E2 -21729.308} C_VEL
LIN {X 0,Y 226.111,Z 384.449,A -85,B 0,C 180,E1 -21730.17,E2 -21730.17} C_VEL
LIN {X 0,Y 220.05,Z 370.324,A -85,B 0,C 180,E1 -21732.351,E2 -21732.351} C_VEL
LIN {X 0,Y 213.976,Z 358.174,A -85,B 0,C 180,E1 -21734.662,E2 -21734.662} C_VEL
LIN {X 0,Y 208.36,Z 348.306,A -85,B 0,C 180,E1 -21736.955,E2 -21736.955} C_VEL
LIN {X 0,Y 205.172,Z 343.155,A -85,B 0,C 180,E1 -21738.342,E2 -21738.342} C_VEL
LIN {X 0,Y 201.887,Z 337.971,A -85,B 0,C 180,E1 -21739.86,E2 -21739.86} C_VEL
LIN {X 0,Y 198.803,Z 333.214,A -85,B 0,C 180,E1 -21741.379,E2 -21741.379} C_VEL
LIN {X 0,Y 195.094,Z 328.183,A -85,B 0,C 180,E1 -21743.31,E2 -21743.31} C_VEL
LIN {X 0,Y 194.265,Z 326.54,A -85,B 0,C 180,E1 -21743.834,E2 -21743.834} C_VEL
LIN {X 0,Y 192.637,Z 321.478,A -85,B 0,C 180,E1 -21748.226,E2 -21748.226} C_VEL
LIN {X 0,Y 192.661,Z 321.474,A -85,B 0,C 180,E1 -21751.692,E2 -21751.692} C_VEL
LIN {X 0,Y 192.707,Z 321.469,A -85,B 0,C 180,E1 -21756.349,E2 -21756.349} C_VEL
LIN {X 0,Y 192.752,Z 321.475,A -85,B 0,C 180,E1 -21761.437,E2 -21761.437} C_VEL
LIN {X 0,Y 192.85,Z 321.453,A -85,B 0,C 180,E1 -21767.37,E2 -21767.37} C_VEL
LIN {X 0,Y 193.07,Z 321.425,A -85,B 0,C 180,E1 -21771.628,E2 -21771.628} C_VEL
LIN {X 0,Y 193.261,Z 321.409,A -85,B 0,C 180,E1 -21777.916,E2 -21777.916} C_VEL
LIN {X 0,Y 193.441,Z 321.379,A -85,B 0,C 180,E1 -21780.001,E2 -21780.001} C_VEL
LIN {X 0,Y 192.976,Z 321.437,A -85,B 0,C 180,E1 -21784.178,E2 -21784.178} C_VEL
LIN {X 0,Y 193.076,Z 321.425,A -85,B 0,C 180,E1 -21788.373,E2 -21788.373} C_VEL
LIN {X 0,Y 192.851,Z 321.453,A -85,B 0,C 180,E1 -21792.631,E2 -21792.631} C_VEL
LIN {X 0,Y 192.779,Z 321.465,A -85,B 0,C 180,E1 -21798.587,E2 -21798.587} C_VEL
LIN {X 0,Y 192.662,Z 321.481,A -85,B 0,C 180,E1 -21804.226,E2 -21804.226} C_VEL
LIN {X 0,Y 192.65,Z 321.591,A -85,B 0,C 180,E1 -21806.764,E2 -21806.764} C_VEL
LIN {X 0,Y 193.522,Z 324.13,A -85,B 0,C 180,E1 -21807.364,E2 -21807.364} C_VEL
LIN {X 0,Y 195.51,Z 326.325,A -85,B 0,C 180,E1 -21808.436,E2 -21808.436} C_VEL
LIN {X 0,Y 196.774,Z 327.334,A -85,B 0,C 180,E1 -21809.065,E2 -21809.065} C_VEL
LIN {X 0,Y 198.747,Z 330.556,A -85,B 0,C 180,E1 -21810.113,E2 -21810.113} C_VEL
LIN {X 0,Y 200.689,Z 332.543,A -85,B 0,C 180,E1 -21811.028,E2 -21811.028} C_VEL
LIN {X 0,Y 203.272,Z 336.139,A -85,B 0,C 180,E1 -21812.243,E2 -21812.243} C_VEL
LIN {X 0,Y 204.705,Z 338.001,A -85,B 0,C 180,E1 -21812.881,E2 -21812.881} C_VEL
LIN {X 0,Y 208.168,Z 342.777,A -85,B 0,C 180,E1 -21814.365,E2 -21814.365} C_VEL
LIN {X 0,Y 213.231,Z 350.152,A -85,B 0,C 180,E1 -21816.39,E2 -21816.39} C_VEL
LIN {X 0,Y 219.512,Z 360.049,A -85,B 0,C 180,E1 -21818.707,E2 -21818.707} C_VEL
LIN {X 0,Y 226.509,Z 372.528,A -85,B 0,C 180,E1 -21821.092,E2 -21821.092} C_VEL
LIN {X 0,Y 228.637,Z 377.176,A -85,B 0,C 180,E1 -21821.806,E2 -21821.806} C_VEL
LIN {X 0,Y 226.031,Z 421.589,A -85,B 0,C 180,E1 -21823.124,E2 -21823.124} C_VEL
LIN {X 0,Y 224.615,Z 434.727,A -85,B 0,C 180,E1 -21823.821,E2 -21823.821} C_VEL
LIN {X 0,Y 222.461,Z 447.79,A -85,B 0,C 180,E1 -21824.861,E2 -21824.861} C_VEL
LIN {X 0,Y 219.447,Z 460.106,A -85,B 0,C 180,E1 -21826.168,E2 -21826.168} C_VEL
LIN {X 0,Y 216.445,Z 470.721,A -85,B 0,C 180,E1 -21827.707,E2 -21827.707} C_VEL
LIN {X 0,Y 213.321,Z 480.68,A -85,B 0,C 180,E1 -21829.582,E2 -21829.582} C_VEL
LIN {X 0,Y 209.807,Z 489.846,A -85,B 0,C 180,E1 -21831.707,E2 -21831.707} C_VEL
LIN {X 0,Y 206.413,Z 497.809,A -85,B 0,C 180,E1 -21834.034,E2 -21834.034} C_VEL
LIN {X 0,Y 202.753,Z 505.525,A -85,B 0,C 180,E1 -21836.913,E2 -21836.913} C_VEL
LIN {X 0,Y 199.039,Z 512.591,A -85,B 0,C 180,E1 -21840.376,E2 -21840.376} C_VEL
LIN {X 0,Y 196.41,Z 517.266,A -85,B 0,C 180,E1 -21843.454,E2 -21843.454} C_VEL
LIN {X 0,Y 194.276,Z 520.746,A -85,B 0,C 180,E1 -21846.553,E2 -21846.553} C_VEL
LIN {X 0,Y 193.122,Z 522.493,A -85,B 0,C 180,E1 -21848.661,E2 -21848.661} C_VEL
LIN {X 0,Y 191.617,Z 524.548,A -85,B 0,C 180,E1 -21852.483,E2 -21852.483} C_VEL
LIN {X 0,Y 190.923,Z 525.216,A -85,B 0,C 180,E1 -21855.069,E2 -21855.069} C_VEL
LIN {X 0,Y 190.266,Z 524.964,A -85,B 0,C 180,E1 -21859.358,E2 -21859.358} C_VEL
LIN {X 0,Y 190.262,Z 524.253,A -85,B 0,C 180,E1 -21861.505,E2 -21861.505} C_VEL
LIN {X 0,Y 190.55,Z 522.358,A -85,B 0,C 180,E1 -21864.776,E2 -21864.776} C_VEL
LIN {X 0,Y 191.018,Z 518.494,A -85,B 0,C 180,E1 -21868.947,E2 -21868.947} C_VEL
LIN {X 0,Y 191.928,Z 514.342,A -85,B 0,C 180,E1 -21872.1,E2 -21872.1} C_VEL
LIN {X 0,Y 193.332,Z 508.034,A -85,B 0,C 180,E1 -21875.739,E2 -21875.739} C_VEL
LIN {X 0,Y 195.088,Z 501.162,A -85,B 0,C 180,E1 -21878.808,E2 -21878.808} C_VEL
LIN {X 0,Y 197.249,Z 492.558,A -85,B 0,C 180,E1 -21881.823,E2 -21881.823} C_VEL
LIN {X 0,Y 199.419,Z 483.739,A -85,B 0,C 180,E1 -21884.283,E2 -21884.283} C_VEL
LIN {X 0,Y 201.623,Z 474.057,A -85,B 0,C 180,E1 -21886.453,E2 -21886.453} C_VEL
LIN {X 0,Y 203.833,Z 463.436,A -85,B 0,C 180,E1 -21888.339,E2 -21888.339} C_VEL
LIN {X 0,Y 205.71,Z 451.599,A -85,B 0,C 180,E1 -21889.979,E2 -21889.979} C_VEL
LIN {X 0,Y 207.318,Z 439.276,A -85,B 0,C 180,E1 -21891.243,E2 -21891.243} C_VEL
LIN {X 0,Y 208.467,Z 426.471,A -85,B 0,C 180,E1 -21892.167,E2 -21892.167} C_VEL
LIN {X 0,Y 209.277,Z 411.432,A -85,B 0,C 180,E1 -21892.784,E2 -21892.784} C_VEL
LIN {X 0,Y 211.513,Z 359.449,A -85,B 0,C 180,E1 -21894.443,E2 -21894.443} C_VEL
LIN {X 0,Y 205.213,Z 345.327,A -85,B 0,C 180,E1 -21896.027,E2 -21896.027} C_VEL
LIN {X 0,Y 197.576,Z 330.851,A -85,B 0,C 180,E1 -21898.008,E2 -21898.008} C_VEL
LIN {X 0,Y 194.142,Z 325.114,A -85,B 0,C 180,E1 -21898.929,E2 -21898.929} C_VEL
LIN {X 0,Y 192.89,Z 322.88,A -85,B 0,C 180,E1 -21899.282,E2 -21899.282} C_VEL
LIN {X 0,Y 192.592,Z 321.492,A -85,B 0,C 180,E1 -21899.435,E2 -21899.435} C_VEL
LIN {X 0,Y 192.599,Z 321.495,A -85,B 0,C 180,E1 -21903.187,E2 -21903.187} C_VEL
LIN {X 0,Y 192.546,Z 321.5,A -85,B 0,C 180,E1 -21908.355,E2 -21908.355} C_VEL
LIN {X 0,Y 192.49,Z 321.503,A -85,B 0,C 180,E1 -21913.094,E2 -21913.094} C_VEL
LIN {X 0,Y 192.488,Z 321.491,A -85,B 0,C 180,E1 -21916.907,E2 -21916.907} C_VEL
LIN {X 0,Y 192.546,Z 321.499,A -85,B 0,C 180,E1 -21921.646,E2 -21921.646} C_VEL
LIN {X 0,Y 192.599,Z 321.48,A -85,B 0,C 180,E1 -21926.813,E2 -21926.813} C_VEL
LIN {X 0,Y 192.624,Z 321.485,A -85,B 0,C 180,E1 -21931.685,E2 -21931.685} C_VEL
LIN {X 0,Y 192.679,Z 321.468,A -85,B 0,C 180,E1 -21936.344,E2 -21936.344} C_VEL
LIN {X 0,Y 192.736,Z 321.472,A -85,B 0,C 180,E1 -21941.459,E2 -21941.459} C_VEL
LIN {X 0,Y 192.753,Z 321.447,A -85,B 0,C 180,E1 -21945.212,E2 -21945.212} C_VEL
LIN {X 0,Y 192.951,Z 321.448,A -85,B 0,C 180,E1 -21949.566,E2 -21949.566} C_VEL
LIN {X 0,Y 192.971,Z 321.427,A -85,B 0,C 180,E1 -21953.727,E2 -21953.727} C_VEL
LIN {X 0,Y 193.235,Z 321.402,A -85,B 0,C 180,E1 -21957.915,E2 -21957.915} C_VEL
LIN {X 0,Y 193.418,Z 321.39,A -85,B 0,C 180,E1 -21959.999,E2 -21959.999} C_VEL
LIN {X 0,Y 192.939,Z 321.435,A -85,B 0,C 180,E1 -21964.177,E2 -21964.177} C_VEL
LIN {X 0,Y 193.029,Z 321.425,A -85,B 0,C 180,E1 -21968.374,E2 -21968.374} C_VEL
LIN {X 0,Y 192.795,Z 321.468,A -85,B 0,C 180,E1 -21972.633,E2 -21972.633} C_VEL
LIN {X 0,Y 192.72,Z 321.478,A -85,B 0,C 180,E1 -21976.962,E2 -21976.962} C_VEL
LIN {X 0,Y 192.587,Z 321.495,A -85,B 0,C 180,E1 -21981.403,E2 -21981.403} C_VEL
LIN {X 0,Y 192.639,Z 321.489,A -85,B 0,C 180,E1 -21984.204,E2 -21984.204} C_VEL
LIN {X 0,Y 192.604,Z 321.497,A -85,B 0,C 180,E1 -21988.864,E2 -21988.864} C_VEL
LIN {X 0,Y 192.598,Z 321.497,A -85,B 0,C 180,E1 -21993.186,E2 -21993.186} C_VEL
LIN {X 0,Y 192.544,Z 321.502,A -85,B 0,C 180,E1 -21998.353,E2 -21998.353} C_VEL
LIN {X 0,Y 192.487,Z 321.509,A -85,B 0,C 180,E1 -22003.092,E2 -22003.092} C_VEL
LIN {X 0,Y 192.565,Z 321.681,A -85,B 0,C 180,E1 -22007.787,E2 -22007.787} C_VEL
LIN {X 0,Y 194.572,Z 329.281,A -85,B 0,C 180,E1 -22011.706,E2 -22011.706} C_VEL
LIN {X 0,Y 201.532,Z 344.65,A -85,B 0,C 180,E1 -22013.668,E2 -22013.668} C_VEL
LIN {X 0,Y 207.269,Z 359.733,A -85,B 0,C 180,E1 -22015.257,E2 -22015.257} C_VEL
LIN {X 0,Y 209.712,Z 382.499,A -85,B 0,C 180,E1 -22016.533,E2 -22016.533} C_VEL
LIN {X 0,Y 210.155,Z 387.618,A -85,B 0,C 180,E1 -22016.798,E2 -22016.798} C_VEL
LIN {X 0,Y 210.183,Z 391.481,A -85,B 0,C 180,E1 -22016.95,E2 -22016.95} C_VEL
LIN {X 0,Y 209.078,Z 397.274,A -85,B 0,C 180,E1 -22017.007,E2 -22017.007} C_VEL
LIN {X 0,Y 203.985,Z 412.486,A -85,B 0,C 180,E1 -22016.821,E2 -22016.821} C_VEL
LIN {X 0,Y 203.042,Z 418.397,A -85,B 0,C 180,E1 -22016.909,E2 -22016.909} C_VEL
LIN {X 0,Y 202.062,Z 439.601,A -85,B 0,C 180,E1 -22017.681,E2 -22017.681} C_VEL
LIN {X 0,Y 200.683,Z 453.146,A -85,B 0,C 180,E1 -22018.53,E2 -22018.53} C_VEL
LIN {X 0,Y 198.77,Z 465.958,A -85,B 0,C 180,E1 -22019.744,E2 -22019.744} C_VEL
LIN {X 0,Y 196.399,Z 478.511,A -85,B 0,C 180,E1 -22021.404,E2 -22021.404} C_VEL
LIN {X 0,Y 193.872,Z 489.701,A -85,B 0,C 180,E1 -22023.345,E2 -22023.345} C_VEL
LIN {X 0,Y 191.439,Z 499.766,A -85,B 0,C 180,E1 -22025.605,E2 -22025.605} C_VEL
LIN {X 0,Y 189.183,Z 509.037,A -85,B 0,C 180,E1 -22028.237,E2 -22028.237} C_VEL
LIN {X 0,Y 187.4,Z 516.444,A -85,B 0,C 180,E1 -22030.842,E2 -22030.842} C_VEL
LIN {X 0,Y 185.589,Z 523.835,A -85,B 0,C 180,E1 -22034.064,E2 -22034.064} C_VEL
LIN {X 0,Y 184.417,Z 528.827,A -85,B 0,C 180,E1 -22036.781,E2 -22036.781} C_VEL
LIN {X 0,Y 183.664,Z 533.682,A -85,B 0,C 180,E1 -22040.083,E2 -22040.083} C_VEL
LIN {X 0,Y 183.287,Z 537.387,A -85,B 0,C 180,E1 -22043.393,E2 -22043.393} C_VEL
LIN {X 0,Y 183.234,Z 539.406,A -85,B 0,C 180,E1 -22045.74,E2 -22045.74} C_VEL
LIN {X 0,Y 183.305,Z 540.738,A -85,B 0,C 180,E1 -22047.801,E2 -22047.801} C_VEL
LIN {X 0,Y 183.43,Z 541.749,A -85,B 0,C 180,E1 -22049.999,E2 -22049.999} C_VEL
LIN {X 0,Y 183.153,Z 542.522,A -85,B 0,C 180,E1 -22053.906,E2 -22053.906} C_VEL
LIN {X 0,Y 183.203,Z 542.339,A -85,B 0,C 180,E1 -22056.607,E2 -22056.607} C_VEL
LIN {X 0,Y 183.933,Z 540.721,A -85,B 0,C 180,E1 -22061.013,E2 -22061.013} C_VEL
LIN {X 0,Y 184.627,Z 539.333,A -85,B 0,C 180,E1 -22063.201,E2 -22063.201} C_VEL
LIN {X 0,Y 186.151,Z 536.435,A -85,B 0,C 180,E1 -22066.447,E2 -22066.447} C_VEL
LIN {X 0,Y 188.346,Z 532.534,A -85,B 0,C 180,E1 -22069.621,E2 -22069.621} C_VEL
LIN {X 0,Y 191.109,Z 527.527,A -85,B 0,C 180,E1 -22072.713,E2 -22072.713} C_VEL
LIN {X 0,Y 194.256,Z 521.264,A -85,B 0,C 180,E1 -22075.73,E2 -22075.73} C_VEL
LIN {X 0,Y 198.092,Z 513.475,A -85,B 0,C 180,E1 -22078.616,E2 -22078.616} C_VEL
LIN {X 0,Y 202.519,Z 503.767,A -85,B 0,C 180,E1 -22081.367,E2 -22081.367} C_VEL
LIN {X 0,Y 206.589,Z 493.751,A -85,B 0,C 180,E1 -22083.559,E2 -22083.559} C_VEL
LIN {X 0,Y 210.125,Z 483.852,A -85,B 0,C 180,E1 -22085.235,E2 -22085.235} C_VEL
LIN {X 0,Y 213.322,Z 473.121,A -85,B 0,C 180,E1 -22086.664,E2 -22086.664} C_VEL
LIN {X 0,Y 216.501,Z 460.198,A -85,B 0,C 180,E1 -22087.932,E2 -22087.932} C_VEL
LIN {X 0,Y 218.773,Z 447.803,A -85,B 0,C 180,E1 -22088.788,E2 -22088.788} C_VEL
LIN {X 0,Y 220.244,Z 434.225,A -85,B 0,C 180,E1 -22089.404,E2 -22089.404} C_VEL
LIN {X 0,Y 222.447,Z 397.154,A -85,B 0,C 180,E1 -22090.516,E2 -22090.516} C_VEL
LIN {X 0,Y 221.224,Z 387.533,A -85,B 0,C 180,E1 -22091.256,E2 -22091.256} C_VEL
LIN {X 0,Y 215.651,Z 374.332,A -85,B 0,C 180,E1 -22093.381,E2 -22093.381} C_VEL
LIN {X 0,Y 210.085,Z 362.954,A -85,B 0,C 180,E1 -22095.623,E2 -22095.623} C_VEL
LIN {X 0,Y 204.399,Z 352.775,A -85,B 0,C 180,E1 -22098.08,E2 -22098.08} C_VEL
LIN {X 0,Y 201.772,Z 348.45,A -85,B 0,C 180,E1 -22099.289,E2 -22099.289} C_VEL
LIN {X 0,Y 198.231,Z 342.821,A -85,B 0,C 180,E1 -22101.019,E2 -22101.019} C_VEL
LIN {X 0,Y 195.134,Z 337.981,A -85,B 0,C 180,E1 -22102.646,E2 -22102.646} C_VEL
LIN {X 0,Y 192.109,Z 333.613,A -85,B 0,C 180,E1 -22104.335,E2 -22104.335} C_VEL
LIN {X 0,Y 191.11,Z 332.117,A -85,B 0,C 180,E1 -22104.928,E2 -22104.928} C_VEL
LIN {X 0,Y 187.122,Z 326.725,A -85,B 0,C 180,E1 -22107.427,E2 -22107.427} C_VEL
LIN {X 0,Y 186.715,Z 325.813,A -85,B 0,C 180,E1 -22107.775,E2 -22107.775} C_VEL
LIN {X 0,Y 185.619,Z 322.353,A -85,B 0,C 180,E1 -22111.29,E2 -22111.29} C_VEL
